   LIN {X 4.730, Y 38.392, Z 10.200} C_DIS
   LIN {X 4.962, Y 37.586, Z 10.200} C_DIS
   LIN {X 5.429, Y 35.866, Z 10.200} C_DIS
   LIN {X 5.472, Y 35.706, Z 10.200} C_DIS
   LIN {X 5.506, Y 35.572, Z 10.200} C_DIS
   LIN {X 6.084, Y 33.263, Z 10.200} C_DIS
   LIN {X 6.346, Y 32.125, Z 10.200} C_DIS
   LIN {X 6.530, Y 31.325, Z 10.200} C_DIS
   LIN {X 7.402, Y 26.882, Z 10.200} C_DIS
   LIN {X 7.443, Y 26.679, Z 10.200} C_DIS
   LIN {X 7.483, Y 26.451, Z 10.200} C_DIS
   LIN {X 7.771, Y 24.714, Z 10.200} C_DIS
   LIN {X 8.198, Y 21.694, Z 10.200} C_DIS
   LIN {X 8.305, Y 20.843, Z 10.200} C_DIS
   LIN {X 8.407, Y 19.968, Z 10.200} C_DIS
   LIN {X 8.478, Y 19.358, Z 10.200} C_DIS
   LIN {X 8.502, Y 19.110, Z 10.200} C_DIS
   LIN {X 8.808, Y 15.682, Z 10.200} C_DIS
   LIN {X 8.841, Y 15.275, Z 10.200} C_DIS
   LIN {X 8.850, Y 15.139, Z 10.200} C_DIS
   LIN {X 8.857, Y 15.004, Z 10.200} C_DIS
   LIN {X 8.864, Y 14.867, Z 10.200} C_DIS
   LIN {X 8.927, Y 13.736, Z 10.200} C_DIS
   LIN {X 9.005, Y 12.397, Z 10.200} C_DIS
   LIN {X 9.017, Y 12.053, Z 10.200} C_DIS
   LIN {X 9.102, Y 8.921, Z 10.200} C_DIS
   LIN {X 9.107, Y 7.373, Z 10.200} C_DIS
   LIN {X 9.109, Y 6.968, Z 10.200} C_DIS
   LIN {X 9.106, Y 6.824, Z 10.200} C_DIS
   LIN {X 9.029, Y 3.343, Z 10.200} C_DIS
   LIN {X 8.935, Y 1.364, Z 10.200} C_DIS
   LIN {X 8.928, Y 1.257, Z 10.200} C_DIS
   LIN {X 8.900, Y 0.914, Z 10.200} C_DIS
   LIN {X 8.633, Y -2.599, Z 10.200} C_DIS
   LIN {X 8.512, Y -3.854, Z 10.200} C_DIS
   LIN {X 8.395, Y -4.942, Z 10.200} C_DIS
   LIN {X 8.356, Y -5.250, Z 10.200} C_DIS
   LIN {X 7.974, Y -8.182, Z 10.200} C_DIS
   LIN {X 7.923, Y -8.524, Z 10.200} C_DIS
   LIN {X 7.807, Y -9.164, Z 10.200} C_DIS
   LIN {X 7.070, Y -13.450, Z 10.200} C_DIS
   LIN {X 6.629, Y -15.636, Z 10.200} C_DIS
   LIN {X 6.073, Y -18.076, Z 10.200} C_DIS
   LIN {X 5.567, Y -20.105, Z 10.200} C_DIS
   LIN {X 5.149, Y -21.676, Z 10.200} C_DIS
   LIN {X 4.625, Y -23.491, Z 10.200} C_DIS
   LIN {X 4.417, Y -24.222, Z 10.200} C_DIS
   LIN {X 4.241, Y -24.798, Z 10.200} C_DIS
   LIN {X 3.838, Y -26.087, Z 10.200} C_DIS
   LIN {X 2.539, Y -28.357, Z 10.200} C_DIS
   LIN {X 1.987, Y -29.326, Z 10.200} C_DIS
   LIN {X 1.547, Y -29.692, Z 10.200} C_DIS
   LIN {X -0.334, Y -31.205, Z 10.200} C_DIS
   LIN {X -2.195, Y -31.910, Z 10.200} C_DIS
   LIN {X -3.063, Y -32.217, Z 10.200} C_DIS
   LIN {X -4.813, Y -32.267, Z 10.200} C_DIS
   LIN {X -5.950, Y -32.313, Z 10.200} C_DIS
   LIN {X -6.218, Y -32.259, Z 10.200} C_DIS
   LIN {X -6.409, Y -32.191, Z 10.200} C_DIS
   LIN {X -9.906, Y -30.751, Z 10.200} C_DIS
   LIN {X -10.167, Y -30.607, Z 10.200} C_DIS
   LIN {X -10.841, Y -30.035, Z 10.200} C_DIS
   LIN {X -11.131, Y -29.776, Z 10.200} C_DIS
   LIN {X -11.194, Y -29.687, Z 10.200} C_DIS
   LIN {X -11.449, Y -29.321, Z 10.200} C_DIS
   LIN {X -12.804, Y -27.467, Z 10.200} C_DIS
   LIN {X -13.363, Y -25.694, Z 10.200} C_DIS
   LIN {X -13.691, Y -24.527, Z 10.200} C_DIS
   LIN {X -13.623, Y -23.242, Z 10.200} C_DIS
   LIN {X -13.562, Y -21.557, Z 10.200} C_DIS
   LIN {X -12.981, Y -20.117, Z 10.200} C_DIS
   LIN {X -12.370, Y -18.619, Z 10.200} C_DIS
   LIN {X -11.694, Y -17.504, Z 10.200} C_DIS
   LIN {X -10.729, Y -15.883, Z 10.200} C_DIS
   LIN {X -8.996, Y -12.598, Z 10.200} C_DIS
   LIN {X -8.678, Y -12.002, Z 10.200} C_DIS
   LIN {X -8.590, Y -11.835, Z 10.200} C_DIS
   LIN {X -8.537, Y -11.731, Z 10.200} C_DIS
   LIN {X -7.939, Y -10.386, Z 10.200} C_DIS
   LIN {X -6.633, Y -7.473, Z 10.200} C_DIS
   LIN {X -6.291, Y -6.580, Z 10.200} C_DIS
   LIN {X -5.258, Y -3.854, Z 10.200} C_DIS
   LIN {X -4.877, Y -2.572, Z 10.200}
   LaserEnd_Ext()
   LIN {X -0.927, Y -30.360, Z 10.200}
   LaserStart_Ext()
   LIN {X -8.228, Y -30.360, Z 10.200}
   LaserEnd_Ext()
   LIN {X -10.092, Y -29.360, Z 10.200}
   LaserStart_Ext()
   LIN {X 0.364, Y -29.360, Z 10.200}
   LaserEnd_Ext()
   LIN {X 1.386, Y -28.360, Z 10.200}
   LaserStart_Ext()
   LIN {X -10.912, Y -28.360, Z 10.200}
   LaserEnd_Ext()
   LIN {X -11.643, Y -27.360, Z 10.200}
   LaserStart_Ext()
   LIN {X 1.957, Y -27.360, Z 10.200}
   LaserEnd_Ext()
   LIN {X 2.530, Y -26.360, Z 10.200}
   LaserStart_Ext()
   LIN {X -12.104, Y -26.360, Z 10.200}
   LaserEnd_Ext()
   LIN {X -12.418, Y -25.360, Z 10.200}
   LaserStart_Ext()
   LIN {X -5.393, Y -25.360, Z 10.200}
   LaserEnd_Ext()
   LIN {X -4.055, Y -25.360, Z 10.200}
   LaserStart_Ext()
   LIN {X 3.018, Y -25.360, Z 10.200}
   LaserEnd_Ext()
   LIN {X 3.329, Y -24.360, Z 10.200}
   LaserStart_Ext()
   LIN {X -2.856, Y -24.360, Z 10.200}
   LaserEnd_Ext()
   LIN {X -6.619, Y -24.360, Z 10.200}
   LaserStart_Ext()
   LIN {X -12.681, Y -24.360, Z 10.200}
   LaserEnd_Ext()
   LIN {X -12.628, Y -23.360, Z 10.200}
   LaserStart_Ext()
   LIN {X -6.894, Y -23.360, Z 10.200}
   LaserEnd_Ext()
   LIN {X -2.671, Y -23.360, Z 10.200}
   LaserStart_Ext()
   LIN {X 3.623, Y -23.360, Z 10.200}
   LaserEnd_Ext()
   LIN {X 3.911, Y -22.360, Z 10.200}
   LaserStart_Ext()
   LIN {X -2.769, Y -22.360, Z 10.200}
   LaserEnd_Ext()
   LIN {X -6.651, Y -22.360, Z 10.200}
   LaserStart_Ext()
   LIN {X -12.591, Y -22.360, Z 10.200}
   LaserEnd_Ext()
   LIN {X -12.405, Y -21.360, Z 10.200}
   LaserStart_Ext()
   LIN {X -5.680, Y -21.360, Z 10.200}
   LaserEnd_Ext()
   LIN {X -3.731, Y -21.360, Z 10.200}
   LaserStart_Ext()
   LIN {X 4.199, Y -21.360, Z 10.200}
   LaserEnd_Ext()
   LIN {X 4.464, Y -20.360, Z 10.200}
   LaserStart_Ext()
   LIN {X -12.000, Y -20.360, Z 10.200}
   LaserEnd_Ext()
   LIN {X -11.592, Y -19.360, Z 10.200}
   LaserStart_Ext()
   LIN {X 4.722, Y -19.360, Z 10.200}
   LaserEnd_Ext()
   LIN {X 4.972, Y -18.360, Z 10.200}
   LaserStart_Ext()
   LIN {X -11.044, Y -18.360, Z 10.200}
   LaserEnd_Ext()
   LIN {X -10.445, Y -17.360, Z 10.200}
   LaserStart_Ext()
   LIN {X 5.211, Y -17.360, Z 10.200}
   LaserEnd_Ext()
   LIN {X 5.439, Y -16.360, Z 10.200}
   LaserStart_Ext()
   LIN {X -9.851, Y -16.360, Z 10.200}
   LaserEnd_Ext()
   LIN {X -9.323, Y -15.360, Z 10.200}
   LaserStart_Ext()
   LIN {X 5.665, Y -15.360, Z 10.200}
   LaserEnd_Ext()
   LIN {X 5.866, Y -14.360, Z 10.200}
   LaserStart_Ext()
   LIN {X -8.795, Y -14.360, Z 10.200}
   LaserEnd_Ext()
   LIN {X -8.268, Y -13.360, Z 10.200}
   LaserStart_Ext()
   LIN {X 6.068, Y -13.360, Z 10.200}
   LaserEnd_Ext()
   LIN {X 6.243, Y -12.360, Z 10.200}
   LaserStart_Ext()
   LIN {X -7.736, Y -12.360, Z 10.200}
   LaserEnd_Ext()
   LIN {X -7.277, Y -11.360, Z 10.200}
   LaserStart_Ext()
   LIN {X 6.415, Y -11.360, Z 10.200}
   LaserEnd_Ext()
   LIN {X 6.587, Y -10.360, Z 10.200}
   LaserStart_Ext()
   LIN {X -6.831, Y -10.360, Z 10.200}
   LaserEnd_Ext()
   LIN {X -6.383, Y -9.360, Z 10.200}
   LaserStart_Ext()
   LIN {X 6.758, Y -9.360, Z 10.200}
   LaserEnd_Ext()
   LIN {X 6.937, Y -8.360, Z 10.200}
   LaserStart_Ext()
   LIN {X -5.935, Y -8.360, Z 10.200}
   LaserEnd_Ext()
   LIN {X -5.519, Y -7.360, Z 10.200}
   LaserStart_Ext()
   LIN {X 7.073, Y -7.360, Z 10.200}
   LaserEnd_Ext()
   LIN {X 7.203, Y -6.360, Z 10.200}
   LaserStart_Ext()
   LIN {X -5.138, Y -6.360, Z 10.200}
   LaserEnd_Ext()
   LIN {X -4.760, Y -5.360, Z 10.200}
   LaserStart_Ext()
   LIN {X 7.333, Y -5.360, Z 10.200}
   LaserEnd_Ext()
   LIN {X 7.452, Y -4.360, Z 10.200}
   LaserStart_Ext()
   LIN {X -4.381, Y -4.360, Z 10.200}
   LaserEnd_Ext()
   LIN {X -4.068, Y -3.360, Z 10.200}
   LaserStart_Ext()
   LIN {X 7.555, Y -3.360, Z 10.200}
   LaserEnd_Ext()
   LIN {X 7.648, Y -2.360, Z 10.200}
   LaserStart_Ext()
   LIN {X -3.759, Y -2.360, Z 10.200}
   LaserEnd_Ext()
   LIN {X -3.437, Y -1.360, Z 10.200}
   LaserStart_Ext()
   LIN {X 7.724, Y -1.360, Z 10.200}
   LaserEnd_Ext()
   LIN {X 7.800, Y -0.360, Z 10.200}
   LaserStart_Ext()
   LIN {X -3.115, Y -0.360, Z 10.200}
   LaserEnd_Ext()
   LIN {X -2.824, Y 0.640, Z 10.200}
   LaserStart_Ext()
   LIN {X 7.876, Y 0.640, Z 10.200}
   LaserEnd_Ext()
   LIN {X 7.947, Y 1.640, Z 10.200}
   LaserStart_Ext()
   LIN {X -2.546, Y 1.640, Z 10.200}
   LaserEnd_Ext()
   LIN {X -2.297, Y 2.640, Z 10.200}
   LaserStart_Ext()
   LIN {X 7.994, Y 2.640, Z 10.200}
   LaserEnd_Ext()
   LIN {X 8.035, Y 3.640, Z 10.200}
   LaserStart_Ext()
   LIN {X -2.063, Y 3.640, Z 10.200}
   LaserEnd_Ext()
   LIN {X -1.857, Y 4.640, Z 10.200}
   LaserStart_Ext()
   LIN {X 8.057, Y 4.640, Z 10.200}
   LaserEnd_Ext()
   LIN {X 8.080, Y 5.640, Z 10.200}
   LaserStart_Ext()
   LIN {X -1.653, Y 5.640, Z 10.200}
   LaserEnd_Ext()
   LIN {X -1.438, Y 6.640, Z 10.200}
   LaserStart_Ext()
   LIN {X 8.102, Y 6.640, Z 10.200}
   LaserEnd_Ext()
   LIN {X 8.107, Y 7.640, Z 10.200}
   LaserStart_Ext()
   LIN {X -1.262, Y 7.640, Z 10.200}
   LaserEnd_Ext()
   LIN {X -1.098, Y 8.640, Z 10.200}
   LaserStart_Ext()
   LIN {X 8.103, Y 8.640, Z 10.200}
   LaserEnd_Ext()
   LIN {X 8.083, Y 9.640, Z 10.200}
   LaserStart_Ext()
   LIN {X -0.945, Y 9.640, Z 10.200}
   LaserEnd_Ext()
   LIN {X -0.820, Y 10.640, Z 10.200}
   LaserStart_Ext()
   LIN {X 8.055, Y 10.640, Z 10.200}
   LaserEnd_Ext()
   LIN {X 8.028, Y 11.640, Z 10.200}
   LaserStart_Ext()
   LIN {X -0.695, Y 11.640, Z 10.200}
   LaserEnd_Ext()
   LIN {X -0.574, Y 12.640, Z 10.200}
   LaserStart_Ext()
   LIN {X 7.989, Y 12.640, Z 10.200}
   LaserEnd_Ext()
   LIN {X 7.931, Y 13.640, Z 10.200}
   LaserStart_Ext()
   LIN {X -0.496, Y 13.640, Z 10.200}
   LaserEnd_Ext()
   LIN {X -0.418, Y 14.640, Z 10.200}
   LaserStart_Ext()
   LIN {X 7.875, Y 14.640, Z 10.200}
   LaserEnd_Ext()
   LIN {X 7.808, Y 15.640, Z 10.200}
   LaserStart_Ext()
   LIN {X -0.340, Y 15.640, Z 10.200}
   LaserEnd_Ext()
   LIN {X -0.276, Y 16.640, Z 10.200}
   LaserStart_Ext()
   LIN {X 7.719, Y 16.640, Z 10.200}
   LaserEnd_Ext()
   LIN {X 7.630, Y 17.640, Z 10.200}
   LaserStart_Ext()
   LIN {X -0.236, Y 17.640, Z 10.200}
   LaserEnd_Ext()
   LIN {X -0.209, Y 18.640, Z 10.200}
   LaserStart_Ext()
   LIN {X 7.540, Y 18.640, Z 10.200}
   LaserEnd_Ext()
   LIN {X 7.439, Y 19.640, Z 10.200}
   LaserStart_Ext()
   LIN {X -0.198, Y 19.640, Z 10.200}
   LaserEnd_Ext()
   LIN {X -0.205, Y 20.640, Z 10.200}
   LaserStart_Ext()
   LIN {X 7.322, Y 20.640, Z 10.200}
   LaserEnd_Ext()
   LIN {X 7.195, Y 21.640, Z 10.200}
   LaserStart_Ext()
   LIN {X -0.229, Y 21.640, Z 10.200}
   LaserEnd_Ext()
   LIN {X -0.254, Y 22.640, Z 10.200}
   LaserStart_Ext()
   LIN {X 7.054, Y 22.640, Z 10.200}
   LaserEnd_Ext()
   LIN {X 6.913, Y 23.640, Z 10.200}
   LaserStart_Ext()
   LIN {X -0.278, Y 23.640, Z 10.200}
   LaserEnd_Ext()
   LIN {X -0.333, Y 24.640, Z 10.200}
   LaserStart_Ext()
   LIN {X 6.769, Y 24.640, Z 10.200}
   LaserEnd_Ext()
   LIN {X 6.604, Y 25.640, Z 10.200}
   LaserStart_Ext()
   LIN {X -0.404, Y 25.640, Z 10.200}
   LaserEnd_Ext()
   LIN {X -0.489, Y 26.640, Z 10.200}
   LaserStart_Ext()
   LIN {X 6.431, Y 26.640, Z 10.200}
   LaserEnd_Ext()
   LIN {X 6.234, Y 27.640, Z 10.200}
   LaserStart_Ext()
   LIN {X -0.590, Y 27.640, Z 10.200}
   LaserEnd_Ext()
   LIN {X -0.692, Y 28.640, Z 10.200}
   LaserStart_Ext()
   LIN {X 6.038, Y 28.640, Z 10.200}
   LaserEnd_Ext()
   LIN {X 5.842, Y 29.640, Z 10.200}
   LaserStart_Ext()
   LIN {X -0.813, Y 29.640, Z 10.200}
   LaserEnd_Ext()
   LIN {X -0.956, Y 30.640, Z 10.200}
   LaserStart_Ext()
   LIN {X 5.646, Y 30.640, Z 10.200}
   LaserEnd_Ext()
   LIN {X 5.431, Y 31.640, Z 10.200}
   LaserStart_Ext()
   LIN {X -1.099, Y 31.640, Z 10.200}
   LaserEnd_Ext()
   LIN {X -1.261, Y 32.640, Z 10.200}
   LaserStart_Ext()
   LIN {X 5.201, Y 32.640, Z 10.200}
   LaserEnd_Ext()
   LIN {X 4.959, Y 33.640, Z 10.200}
   LaserStart_Ext()
   LIN {X -1.441, Y 33.640, Z 10.200}
   LaserEnd_Ext()
   LIN {X -1.627, Y 34.640, Z 10.200}
   LaserStart_Ext()
   LIN {X 4.709, Y 34.640, Z 10.200}
   LaserEnd_Ext()
   LIN {X 4.454, Y 35.640, Z 10.200}
   LaserStart_Ext()
   LIN {X -1.836, Y 35.640, Z 10.200}
   LaserEnd_Ext()
   LIN {X -2.052, Y 36.640, Z 10.200}
   LaserStart_Ext()
   LIN {X 4.182, Y 36.640, Z 10.200}
   LaserEnd_Ext()
   LIN {X 3.906, Y 37.640, Z 10.200}
   LaserStart_Ext()
   LIN {X -2.199, Y 37.640, Z 10.200}
   LaserEnd_Ext()
   LIN {X -2.148, Y 38.640, Z 10.200}
   LaserStart_Ext()
   LIN {X 3.617, Y 38.640, Z 10.200}
   LaserEnd_Ext()
   LIN {X 3.121, Y 39.640, Z 10.200}
   LaserStart_Ext()
   LIN {X -1.702, Y 39.640, Z 10.200}
   LaserEnd_Ext()
   LIN {X -0.132, Y 40.640, Z 10.200}
   LaserStart_Ext()
   LIN {X 1.883, Y 40.640, Z 10.200}
   LaserEnd_Ext()
   LIN {X -6.268, Y -21.991, Z 11.050}
   LaserStart_Ext()
   LIN {X -6.676, Y -23.129, Z 11.050} C_DIS
   LIN {X -6.630, Y -23.393, Z 11.050} C_DIS
   LIN {X -6.422, Y -24.182, Z 11.050} C_DIS
   LIN {X -6.288, Y -24.390, Z 11.050} C_DIS
   LIN {X -6.019, Y -24.701, Z 11.050} C_DIS
   LIN {X -5.700, Y -24.925, Z 11.050} C_DIS
   LIN {X -5.541, Y -25.028, Z 11.050} C_DIS
   LIN {X -5.254, Y -25.113, Z 11.050} C_DIS
   LIN {X -4.893, Y -25.217, Z 11.050} C_DIS
   LIN {X -4.115, Y -25.153, Z 11.050} C_DIS
   LIN {X -3.320, Y -24.726, Z 11.050} C_DIS
   LIN {X -2.743, Y -23.895, Z 11.050} C_DIS
   LIN {X -2.646, Y -22.978, Z 11.050} C_DIS
   LIN {X -2.635, Y -22.876, Z 11.050} C_DIS
   LIN {X -2.683, Y -22.714, Z 11.050} C_DIS
   LIN {X -2.799, Y -22.327, Z 11.050} C_DIS
   LIN {X -2.978, Y -22.045, Z 11.050} C_DIS
   LIN {X -3.106, Y -21.854, Z 11.050} C_DIS
   LIN {X -3.553, Y -21.505, Z 11.050} C_DIS
   LIN {X -3.707, Y -21.381, Z 11.050} C_DIS
   LIN {X -3.910, Y -21.327, Z 11.050} C_DIS
   LIN {X -4.518, Y -21.162, Z 11.050} C_DIS
   LIN {X -4.733, Y -21.182, Z 11.050} C_DIS
   LIN {X -5.193, Y -21.239, Z 11.050} C_DIS
   LIN {X -6.249, Y -21.966, Z 11.050} C_DIS
   LIN {X -6.268, Y -21.991, Z 11.050}
   LaserEnd_Ext()
   LIN {X -1.587, Y 27.145, Z 11.050}
   LaserStart_Ext()
   LIN {X -1.698, Y 28.227, Z 11.050} C_DIS
   LIN {X -1.788, Y 29.112, Z 11.050} C_DIS
   LIN {X -1.997, Y 30.562, Z 11.050} C_DIS
   LIN {X -2.204, Y 31.978, Z 11.050} C_DIS
   LIN {X -2.451, Y 33.326, Z 11.050} C_DIS
   LIN {X -2.629, Y 34.311, Z 11.050} C_DIS
   LIN {X -2.716, Y 34.727, Z 11.050} C_DIS
   LIN {X -2.959, Y 35.877, Z 11.050} C_DIS
   LIN {X -3.169, Y 36.818, Z 11.050} C_DIS
   LIN {X -3.233, Y 37.099, Z 11.050} C_DIS
   LIN {X -3.257, Y 37.673, Z 11.050} C_DIS
   LIN {X -3.305, Y 38.649, Z 11.050} C_DIS
   LIN {X -3.053, Y 39.374, Z 11.050} C_DIS
   LIN {X -2.780, Y 40.095, Z 11.050} C_DIS
   LIN {X -2.141, Y 40.740, Z 11.050} C_DIS
   LIN {X -1.529, Y 41.382, Z 11.050} C_DIS
   LIN {X -0.612, Y 41.638, Z 11.050} C_DIS
   LIN {X 0.767, Y 42.010, Z 11.050} C_DIS
   LIN {X 1.941, Y 41.701, Z 11.050} C_DIS
   LIN {X 2.458, Y 41.562, Z 11.050} C_DIS
   LIN {X 3.056, Y 41.061, Z 11.050} C_DIS
   LIN {X 3.795, Y 40.443, Z 11.050} C_DIS
   LIN {X 4.094, Y 39.860, Z 11.050} C_DIS
   LIN {X 4.465, Y 39.130, Z 11.050} C_DIS
   LIN {X 4.760, Y 38.111, Z 11.050} C_DIS
   LIN {X 4.902, Y 37.627, Z 11.050} C_DIS
   LIN {X 5.021, Y 37.196, Z 11.050} C_DIS
   LIN {X 5.420, Y 35.738, Z 11.050} C_DIS
   LIN {X 5.963, Y 33.578, Z 11.050} C_DIS
   LIN {X 6.076, Y 33.126, Z 11.050} C_DIS
   LIN {X 6.235, Y 32.437, Z 11.050} C_DIS
   LIN {X 6.550, Y 31.068, Z 11.050} C_DIS
   LIN {X 7.293, Y 27.283, Z 11.050} C_DIS
   LIN {X 7.468, Y 26.385, Z 11.050} C_DIS
   LIN {X 7.598, Y 25.570, Z 11.050} C_DIS
   LIN {X 7.815, Y 24.263, Z 11.050} C_DIS
   LIN {X 8.099, Y 22.252, Z 11.050} C_DIS
   LIN {X 8.363, Y 20.166, Z 11.050} C_DIS
   LIN {X 8.494, Y 19.041, Z 11.050} C_DIS
   LIN {X 8.820, Y 15.370, Z 11.050} C_DIS
   LIN {X 8.855, Y 14.892, Z 11.050} C_DIS
   LIN {X 8.997, Y 12.432, Z 11.050} C_DIS
   LIN {X 9.035, Y 11.400, Z 11.050} C_DIS
   LIN {X 9.101, Y 8.956, Z 11.050} C_DIS
   LIN {X 9.107, Y 7.334, Z 11.050} C_DIS
   LIN {X 9.109, Y 6.597, Z 11.050} C_DIS
   LIN {X 9.043, Y 3.619, Z 11.050} C_DIS
   LIN {X 9.029, Y 3.109, Z 11.050} C_DIS
   LIN {X 8.952, Y 1.501, Z 11.050} C_DIS
   LIN {X 8.905, Y 0.693, Z 11.050} C_DIS
   LIN {X 8.689, Y -2.135, Z 11.050} C_DIS
   LIN {X 8.448, Y -4.657, Z 11.050} C_DIS
   LIN {X 8.424, Y -4.872, Z 11.050} C_DIS
   LIN {X 8.310, Y -5.755, Z 11.050} C_DIS
   LIN {X 7.991, Y -8.255, Z 11.050} C_DIS
   LIN {X 7.835, Y -9.263, Z 11.050} C_DIS
   LIN {X 7.198, Y -12.969, Z 11.050} C_DIS
   LIN {X 6.519, Y -16.333, Z 11.050} C_DIS
   LIN {X 6.216, Y -17.665, Z 11.050} C_DIS
   LIN {X 5.381, Y -21.013, Z 11.050} C_DIS
   LIN {X 5.245, Y -21.523, Z 11.050} C_DIS
   LIN {X 5.075, Y -22.112, Z 11.050} C_DIS
   LIN {X 4.493, Y -24.156, Z 11.050} C_DIS
   LIN {X 4.002, Y -25.765, Z 11.050} C_DIS
   LIN {X 3.921, Y -26.025, Z 11.050} C_DIS
   LIN {X 3.659, Y -26.483, Z 11.050} C_DIS
   LIN {X 2.075, Y -29.266, Z 11.050} C_DIS
   LIN {X 0.809, Y -30.317, Z 11.050} C_DIS
   LIN {X -0.198, Y -31.127, Z 11.050} C_DIS
   LIN {X -2.516, Y -32.005, Z 11.050} C_DIS
   LIN {X -2.875, Y -32.148, Z 11.050} C_DIS
   LIN {X -3.148, Y -32.175, Z 11.050} C_DIS
   LIN {X -5.770, Y -32.280, Z 11.050} C_DIS
   LIN {X -6.545, Y -32.125, Z 11.050} C_DIS
   LIN {X -7.097, Y -31.928, Z 11.050} C_DIS
   LIN {X -9.327, Y -31.010, Z 11.050} C_DIS
   LIN {X -9.944, Y -30.671, Z 11.050} C_DIS
   LIN {X -10.472, Y -30.223, Z 11.050} C_DIS
   LIN {X -10.975, Y -29.813, Z 11.050} C_DIS
   LIN {X -11.154, Y -29.620, Z 11.050} C_DIS
   LIN {X -11.482, Y -29.153, Z 11.050} C_DIS
   LIN {X -12.688, Y -27.503, Z 11.050} C_DIS
   LIN {X -13.496, Y -24.937, Z 11.050} C_DIS
   LIN {X -13.597, Y -24.641, Z 11.050} C_DIS
   LIN {X -13.595, Y -24.371, Z 11.050} C_DIS
   LIN {X -13.492, Y -21.533, Z 11.050} C_DIS
   LIN {X -12.309, Y -18.605, Z 11.050} C_DIS
   LIN {X -10.673, Y -15.853, Z 11.050} C_DIS
   LIN {X -9.083, Y -12.840, Z 11.050} C_DIS
   LIN {X -8.631, Y -11.983, Z 11.050} C_DIS
   LIN {X -8.372, Y -11.427, Z 11.050} C_DIS
   LIN {X -6.783, Y -7.883, Z 11.050} C_DIS
   LIN {X -6.017, Y -5.881, Z 11.050} C_DIS
   LIN {X -5.215, Y -3.764, Z 11.050} C_DIS
   LIN {X -4.457, Y -1.215, Z 11.050} C_DIS
   LIN {X -3.867, Y 0.618, Z 11.050} C_DIS
   LIN {X -3.554, Y 1.723, Z 11.050} C_DIS
   LIN {X -3.290, Y 2.781, Z 11.050} C_DIS
   LIN {X -3.188, Y 3.239, Z 11.050} C_DIS
   LIN {X -2.871, Y 4.788, Z 11.050} C_DIS
   LIN {X -2.413, Y 6.861, Z 11.050} C_DIS
   LIN {X -2.071, Y 8.916, Z 11.050} C_DIS
   LIN {X -1.996, Y 9.426, Z 11.050} C_DIS
   LIN {X -1.613, Y 12.426, Z 11.050} C_DIS
   LIN {X -1.540, Y 13.310, Z 11.050} C_DIS
   LIN {X -1.323, Y 16.095, Z 11.050} C_DIS
   LIN {X -1.299, Y 16.648, Z 11.050} C_DIS
   LIN {X -1.268, Y 17.324, Z 11.050} C_DIS
   LIN {X -1.243, Y 18.170, Z 11.050} C_DIS
   LIN {X -1.231, Y 19.188, Z 11.050} C_DIS
   LIN {X -1.229, Y 20.623, Z 11.050} C_DIS
   LIN {X -1.294, Y 23.277, Z 11.050} C_DIS
   LIN {X -1.341, Y 24.101, Z 11.050} C_DIS
   LIN {X -1.403, Y 24.943, Z 11.050} C_DIS
   LIN {X -1.463, Y 25.994, Z 11.050} C_DIS
   LIN {X -1.552, Y 26.799, Z 11.050} C_DIS
   LIN {X -1.587, Y 27.145, Z 11.050}
   LaserEnd_Ext()
   LIN {X 7.602, Y -3.000, Z 11.050}
   LaserStart_Ext()
   LIN {X 7.602, Y 17.784, Z 11.050}
   LaserEnd_Ext()
   LIN {X 6.602, Y 25.467, Z 11.050}
   LaserStart_Ext()
   LIN {X 6.602, Y -10.533, Z 11.050}
   LaserEnd_Ext()
   LIN {X 5.602, Y -15.824, Z 11.050}
   LaserStart_Ext()
   LIN {X 5.602, Y 30.708, Z 11.050}
   LaserEnd_Ext()
   LIN {X 4.602, Y 34.889, Z 11.050}
   LaserStart_Ext()
   LIN {X 4.602, Y -20.003, Z 11.050}
   LaserEnd_Ext()
   LIN {X 3.602, Y -23.634, Z 11.050}
   LaserStart_Ext()
   LIN {X 3.602, Y 38.515, Z 11.050}
   LaserEnd_Ext()
   LIN {X 2.602, Y 40.137, Z 11.050}
   LaserStart_Ext()
   LIN {X 2.602, Y -26.318, Z 11.050}
   LaserEnd_Ext()
   LIN {X 1.602, Y -28.076, Z 11.050}
   LaserStart_Ext()
   LIN {X 1.602, Y 40.756, Z 11.050}
   LaserEnd_Ext()
   LIN {X 0.602, Y 40.930, Z 11.050}
   LaserStart_Ext()
   LIN {X 0.602, Y -29.189, Z 11.050}
   LaserEnd_Ext()
   LIN {X -0.398, Y -30.005, Z 11.050}
   LaserStart_Ext()
   LIN {X -0.398, Y 15.098, Z 11.050}
   LaserEnd_Ext()
   LIN {X -0.398, Y 24.916, Z 11.050}
   LaserStart_Ext()
   LIN {X -0.398, Y 40.660, Z 11.050}
   LaserEnd_Ext()
   LIN {X -1.398, Y 40.070, Z 11.050}
   LaserStart_Ext()
   LIN {X -1.398, Y 33.127, Z 11.050}
   LaserEnd_Ext()
   LIN {X -1.398, Y 6.871, Z 11.050}
   LaserStart_Ext()
   LIN {X -1.398, Y -30.512, Z 11.050}
   LaserEnd_Ext()
   LIN {X -2.398, Y -30.891, Z 11.050}
   LaserStart_Ext()
   LIN {X -2.398, Y -25.160, Z 11.050}
   LaserEnd_Ext()
   LIN {X -2.398, Y -21.150, Z 11.050}
   LaserStart_Ext()
   LIN {X -2.398, Y 2.224, Z 11.050}
   LaserEnd_Ext()
   LIN {X -3.398, Y -1.188, Z 11.050}
   LaserStart_Ext()
   LIN {X -3.398, Y -20.432, Z 11.050}
   LaserEnd_Ext()
   LIN {X -3.398, Y -25.908, Z 11.050}
   LaserStart_Ext()
   LIN {X -3.398, Y -31.184, Z 11.050}
   LaserEnd_Ext()
   LIN {X -4.398, Y -31.224, Z 11.050}
   LaserStart_Ext()
   LIN {X -4.398, Y -26.180, Z 11.050}
   LaserEnd_Ext()
   LIN {X -4.398, Y -20.171, Z 11.050}
   LaserStart_Ext()
   LIN {X -4.398, Y -4.430, Z 11.050}
   LaserEnd_Ext()
   LIN {X -5.398, Y -7.062, Z 11.050}
   LaserStart_Ext()
   LIN {X -5.398, Y -20.261, Z 11.050}
   LaserEnd_Ext()
   LIN {X -5.398, Y -26.112, Z 11.050}
   LaserStart_Ext()
   LIN {X -5.398, Y -31.265, Z 11.050}
   LaserEnd_Ext()
   LIN {X -6.398, Y -31.116, Z 11.050}
   LaserStart_Ext()
   LIN {X -6.398, Y -25.657, Z 11.050}
   LaserEnd_Ext()
   LIN {X -6.398, Y -20.855, Z 11.050}
   LaserStart_Ext()
   LIN {X -6.398, Y -9.469, Z 11.050}
   LaserEnd_Ext()
   LIN {X -7.398, Y -11.700, Z 11.050}
   LaserStart_Ext()
   LIN {X -7.398, Y -22.180, Z 11.050}
   LaserEnd_Ext()
   LIN {X -7.398, Y -24.402, Z 11.050}
   LaserStart_Ext()
   LIN {X -7.398, Y -30.723, Z 11.050}
   LaserEnd_Ext()
   LIN {X -8.398, Y -30.311, Z 11.050}
   LaserStart_Ext()
   LIN {X -8.398, Y -13.685, Z 11.050}
   LaserEnd_Ext()
   LIN {X -9.398, Y -15.580, Z 11.050}
   LaserStart_Ext()
   LIN {X -9.398, Y -29.823, Z 11.050}
   LaserEnd_Ext()
   LIN {X -10.398, Y -28.957, Z 11.050}
   LaserStart_Ext()
   LIN {X -10.398, Y -17.346, Z 11.050}
   LaserEnd_Ext()
   LIN {X -11.398, Y -19.026, Z 11.050}
   LaserStart_Ext()
   LIN {X -11.398, Y -27.573, Z 11.050}
   LaserEnd_Ext()
   LIN {X -12.398, Y -25.095, Z 11.050}
   LaserStart_Ext()
   LIN {X -12.398, Y -21.495, Z 11.050}
   LaserEnd_Ext()
   LIN {X -4.864, Y -25.940, Z 11.900}
   LaserStart_Ext()
   LIN {X -4.243, Y -25.966, Z 11.900} C_DIS
   LIN {X -4.008, Y -25.904, Z 11.900} C_DIS
   LIN {X -3.329, Y -25.702, Z 11.900} C_DIS
   LIN {X -3.119, Y -25.586, Z 11.900} C_DIS
   LIN {X -2.544, Y -24.979, Z 11.900} C_DIS
   LIN {X -1.792, Y -23.871, Z 11.900} C_DIS
   LIN {X -1.766, Y -22.530, Z 11.900} C_DIS
   LIN {X -1.786, Y -22.242, Z 11.900} C_DIS
   LIN {X -1.841, Y -22.124, Z 11.900} C_DIS
   LIN {X -2.889, Y -20.825, Z 11.900} C_DIS
   LIN {X -3.228, Y -20.512, Z 11.900} C_DIS
   LIN {X -3.658, Y -20.387, Z 11.900} C_DIS
   LIN {X -4.266, Y -20.212, Z 11.900} C_DIS
   LIN {X -4.841, Y -20.232, Z 11.900} C_DIS
   LIN {X -5.041, Y -20.247, Z 11.900} C_DIS
   LIN {X -6.009, Y -20.665, Z 11.900} C_DIS
   LIN {X -6.432, Y -20.929, Z 11.900} C_DIS
   LIN {X -7.154, Y -21.901, Z 11.900} C_DIS
   LIN {X -7.307, Y -22.360, Z 11.900} C_DIS
   LIN {X -7.427, Y -23.298, Z 11.900} C_DIS
   LIN {X -6.885, Y -24.784, Z 11.900} C_DIS
   LIN {X -6.758, Y -24.954, Z 11.900} C_DIS
   LIN {X -6.304, Y -25.406, Z 11.900} C_DIS
   LIN {X -6.136, Y -25.512, Z 11.900} C_DIS
   LIN {X -5.822, Y -25.701, Z 11.900} C_DIS
   LIN {X -5.240, Y -25.896, Z 11.900} C_DIS
   LIN {X -5.125, Y -25.932, Z 11.900} C_DIS
   LIN {X -4.864, Y -25.940, Z 11.900}
   LaserEnd_Ext()
   LIN {X 5.376, Y 35.731, Z 11.900}
   LaserStart_Ext()
   LIN {X 4.835, Y 37.695, Z 11.900} C_DIS
   LIN {X 4.532, Y 38.730, Z 11.900} C_DIS
   LIN {X 4.395, Y 39.196, Z 11.900} C_DIS
   LIN {X 4.136, Y 39.699, Z 11.900} C_DIS
   LIN {X 3.722, Y 40.508, Z 11.900} C_DIS
   LIN {X 3.043, Y 41.075, Z 11.900} C_DIS
   LIN {X 2.382, Y 41.624, Z 11.900} C_DIS
   LIN {X 0.705, Y 42.063, Z 11.900} C_DIS
   LIN {X -1.632, Y 41.413, Z 11.900} C_DIS
   LIN {X -2.238, Y 40.795, Z 11.900} C_DIS
   LIN {X -2.800, Y 40.229, Z 11.900} C_DIS
   LIN {X -3.058, Y 39.545, Z 11.900} C_DIS
   LIN {X -3.374, Y 38.685, Z 11.900} C_DIS
   LIN {X -3.345, Y 38.254, Z 11.900} C_DIS
   LIN {X -3.298, Y 37.147, Z 11.900} C_DIS
   LIN {X -3.049, Y 36.049, Z 11.900} C_DIS
   LIN {X -3.022, Y 35.926, Z 11.900} C_DIS
   LIN {X -2.957, Y 35.617, Z 11.900} C_DIS
   LIN {X -2.688, Y 34.360, Z 11.900} C_DIS
   LIN {X -2.390, Y 32.749, Z 11.900} C_DIS
   LIN {X -2.258, Y 32.028, Z 11.900} C_DIS
   LIN {X -2.101, Y 30.957, Z 11.900} C_DIS
   LIN {X -1.835, Y 29.163, Z 11.900} C_DIS
   LIN {X -1.715, Y 27.989, Z 11.900} C_DIS
   LIN {X -1.652, Y 27.374, Z 11.900} C_DIS
   LIN {X -1.493, Y 25.938, Z 11.900} C_DIS
   LIN {X -1.386, Y 24.063, Z 11.900} C_DIS
   LIN {X -1.343, Y 23.467, Z 11.900} C_DIS
   LIN {X -1.309, Y 22.883, Z 11.900} C_DIS
   LIN {X -1.263, Y 21.005, Z 11.900} C_DIS
   LIN {X -1.267, Y 18.546, Z 11.900} C_DIS
   LIN {X -1.275, Y 17.869, Z 11.900} C_DIS
   LIN {X -1.292, Y 17.306, Z 11.900} C_DIS
   LIN {X -1.312, Y 16.856, Z 11.900} C_DIS
   LIN {X -1.353, Y 15.914, Z 11.900} C_DIS
   LIN {X -1.512, Y 13.879, Z 11.900} C_DIS
   LIN {X -1.647, Y 12.244, Z 11.900} C_DIS
   LIN {X -1.932, Y 10.004, Z 11.900} C_DIS
   LIN {X -2.207, Y 8.153, Z 11.900} C_DIS
   LIN {X -2.446, Y 6.715, Z 11.900} C_DIS
   LIN {X -3.187, Y 3.358, Z 11.900} C_DIS
   LIN {X -3.357, Y 2.528, Z 11.900} C_DIS
   LIN {X -3.412, Y 2.283, Z 11.900} C_DIS
   LIN {X -3.553, Y 1.716, Z 11.900} C_DIS
   LIN {X -3.721, Y 1.124, Z 11.900} C_DIS
   LIN {X -4.037, Y 0.141, Z 11.900} C_DIS
   LIN {X -5.172, Y -3.675, Z 11.900} C_DIS
   LIN {X -5.743, Y -5.182, Z 11.900} C_DIS
   LIN {X -6.933, Y -8.292, Z 11.900} C_DIS
   LIN {X -8.083, Y -10.857, Z 11.900} C_DIS
   LIN {X -8.742, Y -12.268, Z 11.900} C_DIS
   LIN {X -9.889, Y -14.445, Z 11.900} C_DIS
   LIN {X -10.616, Y -15.823, Z 11.900} C_DIS
   LIN {X -11.366, Y -17.081, Z 11.900} C_DIS
   LIN {X -12.243, Y -18.567, Z 11.900} C_DIS
   LIN {X -12.741, Y -19.825, Z 11.900} C_DIS
   LIN {X -13.422, Y -21.510, Z 11.900} C_DIS
   LIN {X -13.481, Y -23.132, Z 11.900} C_DIS
   LIN {X -13.496, Y -24.750, Z 11.900} C_DIS
   LIN {X -12.890, Y -26.528, Z 11.900} C_DIS
   LIN {X -12.572, Y -27.539, Z 11.900} C_DIS
   LIN {X -12.096, Y -28.189, Z 11.900} C_DIS
   LIN {X -11.283, Y -29.349, Z 11.900} C_DIS
   LIN {X -10.837, Y -29.829, Z 11.900} C_DIS
   LIN {X -9.873, Y -30.616, Z 11.900} C_DIS
   LIN {X -9.699, Y -30.747, Z 11.900} C_DIS
   LIN {X -9.462, Y -30.877, Z 11.900} C_DIS
   LIN {X -8.749, Y -31.269, Z 11.900} C_DIS
   LIN {X -7.786, Y -31.665, Z 11.900} C_DIS
   LIN {X -6.872, Y -31.991, Z 11.900} C_DIS
   LIN {X -5.590, Y -32.248, Z 11.900} C_DIS
   LIN {X -4.181, Y -32.192, Z 11.900} C_DIS
   LIN {X -2.535, Y -32.031, Z 11.900} C_DIS
   LIN {X -0.370, Y -31.166, Z 11.900} C_DIS
   LIN {X -0.062, Y -31.049, Z 11.900} C_DIS
   LIN {X 0.072, Y -30.942, Z 11.900} C_DIS
   LIN {X 2.163, Y -29.206, Z 11.900} C_DIS
   LIN {X 3.515, Y -26.830, Z 11.900} C_DIS
   LIN {X 4.001, Y -25.960, Z 11.900} C_DIS
   LIN {X 4.145, Y -25.480, Z 11.900} C_DIS
   LIN {X 4.569, Y -24.089, Z 11.900} C_DIS
   LIN {X 5.183, Y -21.932, Z 11.900} C_DIS
   LIN {X 5.372, Y -21.237, Z 11.900} C_DIS
   LIN {X 6.080, Y -18.371, Z 11.900} C_DIS
   LIN {X 6.358, Y -17.254, Z 11.900} C_DIS
   LIN {X 6.410, Y -17.030, Z 11.900} C_DIS
   LIN {X 7.326, Y -12.488, Z 11.900} C_DIS
   LIN {X 7.671, Y -10.477, Z 11.900} C_DIS
   LIN {X 8.043, Y -8.071, Z 11.900} C_DIS
   LIN {X 8.384, Y -5.405, Z 11.900} C_DIS
   LIN {X 8.483, Y -4.496, Z 11.900} C_DIS
   LIN {X 8.568, Y -3.531, Z 11.900} C_DIS
   LIN {X 8.746, Y -1.671, Z 11.900} C_DIS
   LIN {X 8.873, Y -0.004, Z 11.900} C_DIS
   LIN {X 8.973, Y 1.704, Z 11.900} C_DIS
   LIN {X 9.030, Y 2.901, Z 11.900} C_DIS
   LIN {X 9.060, Y 3.981, Z 11.900} C_DIS
   LIN {X 9.110, Y 6.206, Z 11.900} C_DIS
   LIN {X 9.104, Y 7.826, Z 11.900} C_DIS
   LIN {X 9.100, Y 8.992, Z 11.900} C_DIS
   LIN {X 9.053, Y 10.747, Z 11.900} C_DIS
   LIN {X 8.989, Y 12.467, Z 11.900} C_DIS
   LIN {X 8.886, Y 14.247, Z 11.900} C_DIS
   LIN {X 8.776, Y 15.761, Z 11.900} C_DIS
   LIN {X 8.523, Y 18.615, Z 11.900} C_DIS
   LIN {X 8.421, Y 19.490, Z 11.900} C_DIS
   LIN {X 8.001, Y 22.811, Z 11.900} C_DIS
   LIN {X 7.859, Y 23.812, Z 11.900} C_DIS
   LIN {X 7.751, Y 24.463, Z 11.900} C_DIS
   LIN {X 7.477, Y 26.172, Z 11.900} C_DIS
   LIN {X 7.111, Y 28.054, Z 11.900} C_DIS
   LIN {X 6.571, Y 30.811, Z 11.900} C_DIS
   LIN {X 6.123, Y 32.749, Z 11.900} C_DIS
   LIN {X 6.039, Y 33.118, Z 11.900} C_DIS
   LIN {X 5.376, Y 35.731, Z 11.900}
   LaserEnd_Ext()
   LIN {X 2.144, Y 40.522, Z 11.900}
   LaserStart_Ext()
   LIN {X -1.105, Y 40.522, Z 11.900}
   LaserEnd_Ext()
   LIN {X -1.998, Y 39.522, Z 11.900}
   LaserStart_Ext()
   LIN {X 3.103, Y 39.522, Z 11.900}
   LaserEnd_Ext()
   LIN {X 3.551, Y 38.522, Z 11.900}
   LaserStart_Ext()
   LIN {X -2.361, Y 38.522, Z 11.900}
   LaserEnd_Ext()
   LIN {X -2.313, Y 37.522, Z 11.900}
   LaserStart_Ext()
   LIN {X 3.844, Y 37.522, Z 11.900}
   LaserEnd_Ext()
   LIN {X 4.122, Y 36.522, Z 11.900}
   LaserStart_Ext()
   LIN {X -2.131, Y 36.522, Z 11.900}
   LaserEnd_Ext()
   LIN {X -1.914, Y 35.522, Z 11.900}
   LaserStart_Ext()
   LIN {X 4.398, Y 35.522, Z 11.900}
   LaserEnd_Ext()
   LIN {X 4.651, Y 34.522, Z 11.900}
   LaserStart_Ext()
   LIN {X -1.701, Y 34.522, Z 11.900}
   LaserEnd_Ext()
   LIN {X -1.516, Y 33.522, Z 11.900}
   LaserStart_Ext()
   LIN {X 4.905, Y 33.522, Z 11.900}
   LaserEnd_Ext()
   LIN {X 5.149, Y 32.522, Z 11.900}
   LaserStart_Ext()
   LIN {X -1.332, Y 32.522, Z 11.900}
   LaserEnd_Ext()
   LIN {X -1.173, Y 31.522, Z 11.900}
   LaserStart_Ext()
   LIN {X 5.380, Y 31.522, Z 11.900}
   LaserEnd_Ext()
   LIN {X 5.608, Y 30.522, Z 11.900}
   LaserStart_Ext()
   LIN {X -1.025, Y 30.522, Z 11.900}
   LaserEnd_Ext()
   LIN {X -0.877, Y 29.522, Z 11.900}
   LaserStart_Ext()
   LIN {X 5.804, Y 29.522, Z 11.900}
   LaserEnd_Ext()
   LIN {X 6.001, Y 28.522, Z 11.900}
   LaserStart_Ext()
   LIN {X -0.764, Y 28.522, Z 11.900}
   LaserEnd_Ext()
   LIN {X -0.662, Y 27.522, Z 11.900}
   LaserStart_Ext()
   LIN {X 6.196, Y 27.522, Z 11.900}
   LaserEnd_Ext()
   LIN {X 6.391, Y 26.522, Z 11.900}
   LaserStart_Ext()
   LIN {X -0.552, Y 26.522, Z 11.900}
   LaserEnd_Ext()
   LIN {X -0.468, Y 25.522, Z 11.900}
   LaserStart_Ext()
   LIN {X 6.569, Y 25.522, Z 11.900}
   LaserEnd_Ext()
   LIN {X 6.729, Y 24.522, Z 11.900}
   LaserStart_Ext()
   LIN {X -0.410, Y 24.522, Z 11.900}
   LaserEnd_Ext()
   LIN {X -0.344, Y 23.522, Z 11.900}
   LaserStart_Ext()
   LIN {X 6.890, Y 23.522, Z 11.900}
   LaserEnd_Ext()
   LIN {X 7.029, Y 22.522, Z 11.900}
   LaserStart_Ext()
   LIN {X -0.300, Y 22.522, Z 11.900}
   LaserEnd_Ext()
   LIN {X -0.275, Y 21.522, Z 11.900}
   LaserStart_Ext()
   LIN {X 7.156, Y 21.522, Z 11.900}
   LaserEnd_Ext()
   LIN {X 7.282, Y 20.522, Z 11.900}
   LaserStart_Ext()
   LIN {X -0.264, Y 20.522, Z 11.900}
   LaserEnd_Ext()
   LIN {X -0.265, Y 19.522, Z 11.900}
   LaserStart_Ext()
   LIN {X 7.409, Y 19.522, Z 11.900}
   LaserEnd_Ext()
   LIN {X 7.527, Y 18.522, Z 11.900}
   LaserStart_Ext()
   LIN {X -0.267, Y 18.522, Z 11.900}
   LaserEnd_Ext()
   LIN {X -0.285, Y 17.522, Z 11.900}
   LaserStart_Ext()
   LIN {X 7.616, Y 17.522, Z 11.900}
   LaserEnd_Ext()
   LIN {X 7.705, Y 16.522, Z 11.900}
   LaserStart_Ext()
   LIN {X -0.326, Y 16.522, Z 11.900}
   LaserEnd_Ext()
   LIN {X -0.381, Y 15.522, Z 11.900}
   LaserStart_Ext()
   LIN {X 7.791, Y 15.522, Z 11.900}
   LaserEnd_Ext()
   LIN {X 7.864, Y 14.522, Z 11.900}
   LaserStart_Ext()
   LIN {X -0.459, Y 14.522, Z 11.900}
   LaserEnd_Ext()
   LIN {X -0.538, Y 13.522, Z 11.900}
   LaserStart_Ext()
   LIN {X 7.927, Y 13.522, Z 11.900}
   LaserEnd_Ext()
   LIN {X 7.985, Y 12.522, Z 11.900}
   LaserStart_Ext()
   LIN {X -0.620, Y 12.522, Z 11.900}
   LaserEnd_Ext()
   LIN {X -0.731, Y 11.522, Z 11.900}
   LaserStart_Ext()
   LIN {X 8.024, Y 11.522, Z 11.900}
   LaserEnd_Ext()
   LIN {X 8.059, Y 10.522, Z 11.900}
   LaserStart_Ext()
   LIN {X -0.858, Y 10.522, Z 11.900}
   LaserEnd_Ext()
   LIN {X -0.993, Y 9.522, Z 11.900}
   LaserStart_Ext()
   LIN {X 8.086, Y 9.522, Z 11.900}
   LaserEnd_Ext()
   LIN {X 8.102, Y 8.522, Z 11.900}
   LaserStart_Ext()
   LIN {X -1.141, Y 8.522, Z 11.900}
   LaserEnd_Ext()
   LIN {X -1.298, Y 7.522, Z 11.900}
   LaserStart_Ext()
   LIN {X 8.105, Y 7.522, Z 11.900}
   LaserEnd_Ext()
   LIN {X 8.109, Y 6.522, Z 11.900}
   LaserStart_Ext()
   LIN {X -1.465, Y 6.522, Z 11.900}
   LaserEnd_Ext()
   LIN {X -1.686, Y 5.522, Z 11.900}
   LaserStart_Ext()
   LIN {X 8.094, Y 5.522, Z 11.900}
   LaserEnd_Ext()
   LIN {X 8.072, Y 4.522, Z 11.900}
   LaserStart_Ext()
   LIN {X -1.906, Y 4.522, Z 11.900}
   LaserEnd_Ext()
   LIN {X -2.127, Y 3.522, Z 11.900}
   LaserStart_Ext()
   LIN {X 8.047, Y 3.522, Z 11.900}
   LaserEnd_Ext()
   LIN {X 8.011, Y 2.522, Z 11.900}
   LaserStart_Ext()
   LIN {X -2.338, Y 2.522, Z 11.900}
   LaserEnd_Ext()
   LIN {X -2.571, Y 1.522, Z 11.900}
   LaserStart_Ext()
   LIN {X 7.961, Y 1.522, Z 11.900}
   LaserEnd_Ext()
   LIN {X 7.902, Y 0.522, Z 11.900}
   LaserStart_Ext()
   LIN {X -2.864, Y 0.522, Z 11.900}
   LaserEnd_Ext()
   LIN {X -3.178, Y -0.478, Z 11.900}
   LaserStart_Ext()
   LIN {X 7.834, Y -0.478, Z 11.900}
   LaserEnd_Ext()
   LIN {X 7.758, Y -1.478, Z 11.900}
   LaserStart_Ext()
   LIN {X -3.475, Y -1.478, Z 11.900}
   LaserEnd_Ext()
   LIN {X -3.773, Y -2.478, Z 11.900}
   LaserStart_Ext()
   LIN {X 7.664, Y -2.478, Z 11.900}
   LaserEnd_Ext()
   LIN {X 7.569, Y -3.478, Z 11.900}
   LaserStart_Ext()
   LIN {X -4.070, Y -3.478, Z 11.900}
   LaserEnd_Ext()
   LIN {X -4.407, Y -4.478, Z 11.900}
   LaserStart_Ext()
   LIN {X 7.479, Y -4.478, Z 11.900}
   LaserEnd_Ext()
   LIN {X 7.366, Y -5.478, Z 11.900}
   LaserStart_Ext()
   LIN {X -4.786, Y -5.478, Z 11.900}
   LaserEnd_Ext()
   LIN {X -5.168, Y -6.478, Z 11.900}
   LaserStart_Ext()
   LIN {X 7.239, Y -6.478, Z 11.900}
   LaserEnd_Ext()
   LIN {X 7.111, Y -7.478, Z 11.900}
   LaserStart_Ext()
   LIN {X -5.551, Y -7.478, Z 11.900}
   LaserEnd_Ext()
   LIN {X -5.934, Y -8.478, Z 11.900}
   LaserStart_Ext()
   LIN {X 6.968, Y -8.478, Z 11.900}
   LaserEnd_Ext()
   LIN {X 6.814, Y -9.478, Z 11.900}
   LaserStart_Ext()
   LIN {X -6.369, Y -9.478, Z 11.900}
   LaserEnd_Ext()
   LIN {X -6.817, Y -10.478, Z 11.900}
   LaserStart_Ext()
   LIN {X 6.656, Y -10.478, Z 11.900}
   LaserEnd_Ext()
   LIN {X 6.484, Y -11.478, Z 11.900}
   LaserStart_Ext()
   LIN {X -7.269, Y -11.478, Z 11.900}
   LaserEnd_Ext()
   LIN {X -7.736, Y -12.478, Z 11.900}
   LaserStart_Ext()
   LIN {X 6.307, Y -12.478, Z 11.900}
   LaserEnd_Ext()
   LIN {X 6.106, Y -13.478, Z 11.900}
   LaserStart_Ext()
   LIN {X -8.249, Y -13.478, Z 11.900}
   LaserEnd_Ext()
   LIN {X -8.776, Y -14.478, Z 11.900}
   LaserStart_Ext()
   LIN {X 5.904, Y -14.478, Z 11.900}
   LaserEnd_Ext()
   LIN {X 5.702, Y -15.478, Z 11.900}
   LaserStart_Ext()
   LIN {X -9.304, Y -15.478, Z 11.900}
   LaserEnd_Ext()
   LIN {X -9.843, Y -16.478, Z 11.900}
   LaserStart_Ext()
   LIN {X 5.501, Y -16.478, Z 11.900}
   LaserEnd_Ext()
   LIN {X 5.272, Y -17.478, Z 11.900}
   LaserStart_Ext()
   LIN {X -10.438, Y -17.478, Z 11.900}
   LaserEnd_Ext()
   LIN {X -11.029, Y -18.478, Z 11.900}
   LaserStart_Ext()
   LIN {X 5.023, Y -18.478, Z 11.900}
   LaserEnd_Ext()
   LIN {X 4.776, Y -19.478, Z 11.900}
   LaserStart_Ext()
   LIN {X -3.201, Y -19.478, Z 11.900}
   LaserEnd_Ext()
   LIN {X -5.784, Y -19.478, Z 11.900}
   LaserStart_Ext()
   LIN {X -11.528, Y -19.478, Z 11.900}
   LaserEnd_Ext()
   LIN {X -11.927, Y -20.478, Z 11.900}
   LaserStart_Ext()
   LIN {X -7.343, Y -20.478, Z 11.900}
   LaserEnd_Ext()
   LIN {X -1.884, Y -20.478, Z 11.900}
   LaserStart_Ext()
   LIN {X 4.529, Y -20.478, Z 11.900}
   LaserEnd_Ext()
   LIN {X 4.270, Y -21.478, Z 11.900}
   LaserStart_Ext()
   LIN {X -1.077, Y -21.478, Z 11.900}
   LaserEnd_Ext()
   LIN {X -8.059, Y -21.478, Z 11.900}
   LaserStart_Ext()
   LIN {X -12.331, Y -21.478, Z 11.900}
   LaserEnd_Ext()
   LIN {X -12.456, Y -22.478, Z 11.900}
   LaserStart_Ext()
   LIN {X -8.330, Y -22.478, Z 11.900}
   LaserEnd_Ext()
   LIN {X -0.768, Y -22.478, Z 11.900}
   LaserStart_Ext()
   LIN {X 3.988, Y -22.478, Z 11.900}
   LaserEnd_Ext()
   LIN {X 3.703, Y -23.478, Z 11.900}
   LaserStart_Ext()
   LIN {X -0.784, Y -23.478, Z 11.900}
   LaserEnd_Ext()
   LIN {X -8.409, Y -23.478, Z 11.900}
   LaserStart_Ext()
   LIN {X -12.484, Y -23.478, Z 11.900}
   LaserEnd_Ext()
   LIN {X -12.494, Y -24.478, Z 11.900}
   LaserStart_Ext()
   LIN {X -8.061, Y -24.478, Z 11.900}
   LaserEnd_Ext()
   LIN {X -0.996, Y -24.478, Z 11.900}
   LaserStart_Ext()
   LIN {X 3.405, Y -24.478, Z 11.900}
   LaserEnd_Ext()
   LIN {X 3.102, Y -25.478, Z 11.900}
   LaserStart_Ext()
   LIN {X -1.674, Y -25.478, Z 11.900}
   LaserEnd_Ext()
   LIN {X -7.638, Y -25.478, Z 11.900}
   LaserStart_Ext()
   LIN {X -12.191, Y -25.478, Z 11.900}
   LaserEnd_Ext()
   LIN {X -11.857, Y -26.478, Z 11.900}
   LaserStart_Ext()
   LIN {X -6.469, Y -26.478, Z 11.900}
   LaserEnd_Ext()
   LIN {X -2.666, Y -26.478, Z 11.900}
   LaserStart_Ext()
   LIN {X 2.565, Y -26.478, Z 11.900}
   LaserEnd_Ext()
   LIN {X 1.996, Y -27.478, Z 11.900}
   LaserStart_Ext()
   LIN {X -11.377, Y -27.478, Z 11.900}
   LaserEnd_Ext()
   LIN {X -10.672, Y -28.478, Z 11.900}
   LaserStart_Ext()
   LIN {X 1.427, Y -28.478, Z 11.900}
   LaserEnd_Ext()
   LIN {X 0.269, Y -29.478, Z 11.900}
   LaserStart_Ext()
   LIN {X -9.685, Y -29.478, Z 11.900}
   LaserEnd_Ext()
   LIN {X -8.042, Y -30.478, Z 11.900}
   LaserStart_Ext()
   LIN {X -1.344, Y -30.478, Z 11.900}
   LaserEnd_Ext()
   LIN {X -3.075, Y -19.551, Z 12.750}
   LaserStart_Ext()
   LIN {X -4.112, Y -19.254, Z 12.750} C_DIS
   LIN {X -4.898, Y -19.398, Z 12.750} C_DIS
   LIN {X -5.566, Y -19.452, Z 12.750} C_DIS
   LIN {X -6.432, Y -19.847, Z 12.750} C_DIS
   LIN {X -7.078, Y -20.379, Z 12.750} C_DIS
   LIN {X -7.796, Y -21.370, Z 12.750} C_DIS
   LIN {X -8.031, Y -21.981, Z 12.750} C_DIS
   LIN {X -8.177, Y -23.359, Z 12.750} C_DIS
   LIN {X -8.148, Y -23.616, Z 12.750} C_DIS
   LIN {X -8.036, Y -23.929, Z 12.750} C_DIS
   LIN {X -7.670, Y -24.935, Z 12.750} C_DIS
   LIN {X -7.348, Y -25.364, Z 12.750} C_DIS
   LIN {X -7.191, Y -25.580, Z 12.750} C_DIS
   LIN {X -6.785, Y -25.924, Z 12.750} C_DIS
   LIN {X -6.583, Y -26.097, Z 12.750} C_DIS
   LIN {X -6.100, Y -26.375, Z 12.750} C_DIS
   LIN {X -5.325, Y -26.634, Z 12.750} C_DIS
   LIN {X -5.196, Y -26.673, Z 12.750} C_DIS
   LIN {X -4.404, Y -26.718, Z 12.750} C_DIS
   LIN {X -4.211, Y -26.727, Z 12.750} C_DIS
   LIN {X -3.910, Y -26.684, Z 12.750} C_DIS
   LIN {X -3.278, Y -26.527, Z 12.750} C_DIS
   LIN {X -2.758, Y -26.308, Z 12.750} C_DIS
   LIN {X -2.495, Y -26.164, Z 12.750} C_DIS
   LIN {X -2.307, Y -26.037, Z 12.750} C_DIS
   LIN {X -0.994, Y -24.003, Z 12.750} C_DIS
   LIN {X -0.824, Y -23.790, Z 12.750} C_DIS
   LIN {X -0.769, Y -23.474, Z 12.750} C_DIS
   LIN {X -0.857, Y -22.635, Z 12.750} C_DIS
   LIN {X -0.920, Y -21.746, Z 12.750} C_DIS
   LIN {X -1.082, Y -21.396, Z 12.750} C_DIS
   LIN {X -1.346, Y -20.903, Z 12.750} C_DIS
   LIN {X -2.504, Y -19.831, Z 12.750} C_DIS
   LIN {X -2.753, Y -19.640, Z 12.750} C_DIS
   LIN {X -3.075, Y -19.551, Z 12.750}
   LaserEnd_Ext()
   LIN {X 4.417, Y -24.771, Z 12.750}
   LaserStart_Ext()
   LIN {X 4.645, Y -24.022, Z 12.750} C_DIS
   LIN {X 4.976, Y -22.862, Z 12.750} C_DIS
   LIN {X 5.527, Y -20.830, Z 12.750} C_DIS
   LIN {X 6.251, Y -17.898, Z 12.750} C_DIS
   LIN {X 6.452, Y -17.028, Z 12.750} C_DIS
   LIN {X 7.270, Y -12.913, Z 12.750} C_DIS
   LIN {X 7.453, Y -12.006, Z 12.750} C_DIS
   LIN {X 7.508, Y -11.690, Z 12.750} C_DIS
   LIN {X 8.096, Y -7.887, Z 12.750} C_DIS
   LIN {X 8.320, Y -6.135, Z 12.750} C_DIS
   LIN {X 8.551, Y -4.020, Z 12.750} C_DIS
   LIN {X 8.749, Y -1.773, Z 12.750} C_DIS
   LIN {X 8.803, Y -1.208, Z 12.750} C_DIS
   LIN {X 8.842, Y -0.701, Z 12.750} C_DIS
   LIN {X 8.994, Y 1.906, Z 12.750} C_DIS
   LIN {X 9.032, Y 2.693, Z 12.750} C_DIS
   LIN {X 9.078, Y 4.343, Z 12.750} C_DIS
   LIN {X 9.110, Y 5.815, Z 12.750} C_DIS
   LIN {X 9.102, Y 8.319, Z 12.750} C_DIS
   LIN {X 9.099, Y 9.027, Z 12.750} C_DIS
   LIN {X 9.070, Y 10.094, Z 12.750} C_DIS
   LIN {X 8.982, Y 12.502, Z 12.750} C_DIS
   LIN {X 8.918, Y 13.602, Z 12.750} C_DIS
   LIN {X 8.732, Y 16.151, Z 12.750} C_DIS
   LIN {X 8.552, Y 18.188, Z 12.750} C_DIS
   LIN {X 8.479, Y 18.813, Z 12.750} C_DIS
   LIN {X 7.905, Y 23.343, Z 12.750} C_DIS
   LIN {X 7.487, Y 25.959, Z 12.750} C_DIS
   LIN {X 6.930, Y 28.825, Z 12.750} C_DIS
   LIN {X 6.591, Y 30.553, Z 12.750} C_DIS
   LIN {X 6.012, Y 33.061, Z 12.750} C_DIS
   LIN {X 5.827, Y 33.798, Z 12.750} C_DIS
   LIN {X 5.290, Y 35.891, Z 12.750} C_DIS
   LIN {X 4.824, Y 37.567, Z 12.750} C_DIS
   LIN {X 4.767, Y 37.767, Z 12.750} C_DIS
   LIN {X 4.696, Y 38.007, Z 12.750} C_DIS
   LIN {X 4.325, Y 39.262, Z 12.750} C_DIS
   LIN {X 3.881, Y 40.124, Z 12.750} C_DIS
   LIN {X 3.648, Y 40.572, Z 12.750} C_DIS
   LIN {X 2.882, Y 41.206, Z 12.750} C_DIS
   LIN {X 2.306, Y 41.685, Z 12.750} C_DIS
   LIN {X 1.933, Y 41.782, Z 12.750} C_DIS
   LIN {X 0.613, Y 42.124, Z 12.750} C_DIS
   LIN {X -0.912, Y 41.628, Z 12.750} C_DIS
   LIN {X -1.845, Y 41.365, Z 12.750} C_DIS
   LIN {X -2.406, Y 40.794, Z 12.750} C_DIS
   LIN {X -2.903, Y 40.221, Z 12.750} C_DIS
   LIN {X -3.162, Y 39.394, Z 12.750} C_DIS
   LIN {X -3.460, Y 38.581, Z 12.750} C_DIS
   LIN {X -3.381, Y 37.401, Z 12.750} C_DIS
   LIN {X -3.363, Y 37.194, Z 12.750} C_DIS
   LIN {X -3.330, Y 37.053, Z 12.750} C_DIS
   LIN {X -3.084, Y 35.974, Z 12.750} C_DIS
   LIN {X -2.807, Y 34.693, Z 12.750} C_DIS
   LIN {X -2.747, Y 34.410, Z 12.750} C_DIS
   LIN {X -2.658, Y 33.930, Z 12.750} C_DIS
   LIN {X -2.311, Y 32.078, Z 12.750} C_DIS
   LIN {X -2.051, Y 30.354, Z 12.750} C_DIS
   LIN {X -1.882, Y 29.214, Z 12.750} C_DIS
   LIN {X -1.843, Y 28.834, Z 12.750} C_DIS
   LIN {X -1.752, Y 27.948, Z 12.750} C_DIS
   LIN {X -1.523, Y 25.881, Z 12.750} C_DIS
   LIN {X -1.369, Y 23.183, Z 12.750} C_DIS
   LIN {X -1.344, Y 22.833, Z 12.750} C_DIS
   LIN {X -1.324, Y 22.490, Z 12.750} C_DIS
   LIN {X -1.297, Y 21.386, Z 12.750} C_DIS
   LIN {X -1.302, Y 17.905, Z 12.750} C_DIS
   LIN {X -1.306, Y 17.567, Z 12.750} C_DIS
   LIN {X -1.315, Y 17.287, Z 12.750} C_DIS
   LIN {X -1.325, Y 17.063, Z 12.750} C_DIS
   LIN {X -1.383, Y 15.732, Z 12.750} C_DIS
   LIN {X -1.484, Y 14.447, Z 12.750} C_DIS
   LIN {X -1.680, Y 12.063, Z 12.750} C_DIS
   LIN {X -1.869, Y 10.581, Z 12.750} C_DIS
   LIN {X -2.342, Y 7.390, Z 12.750} C_DIS
   LIN {X -2.479, Y 6.569, Z 12.750} C_DIS
   LIN {X -3.503, Y 1.929, Z 12.750} C_DIS
   LIN {X -3.526, Y 1.818, Z 12.750} C_DIS
   LIN {X -3.552, Y 1.709, Z 12.750} C_DIS
   LIN {X -3.617, Y 1.498, Z 12.750} C_DIS
   LIN {X -5.129, Y -3.585, Z 12.750} C_DIS
   LIN {X -5.469, Y -4.483, Z 12.750} C_DIS
   LIN {X -7.084, Y -8.702, Z 12.750} C_DIS
   LIN {X -7.794, Y -10.286, Z 12.750} C_DIS
   LIN {X -8.853, Y -12.554, Z 12.750} C_DIS
   LIN {X -10.496, Y -15.671, Z 12.750} C_DIS
   LIN {X -10.564, Y -15.799, Z 12.750} C_DIS
   LIN {X -10.662, Y -15.969, Z 12.750} C_DIS
   LIN {X -12.181, Y -18.540, Z 12.750} C_DIS
   LIN {X -13.181, Y -21.064, Z 12.750} C_DIS
   LIN {X -13.352, Y -21.487, Z 12.750} C_DIS
   LIN {X -13.367, Y -21.894, Z 12.750} C_DIS
   LIN {X -13.395, Y -24.859, Z 12.750} C_DIS
   LIN {X -12.575, Y -27.267, Z 12.750} C_DIS
   LIN {X -12.459, Y -27.567, Z 12.750} C_DIS
   LIN {X -12.265, Y -27.861, Z 12.750} C_DIS
   LIN {X -11.411, Y -29.078, Z 12.750} C_DIS
   LIN {X -10.700, Y -29.845, Z 12.750} C_DIS
   LIN {X -10.411, Y -30.081, Z 12.750} C_DIS
   LIN {X -9.370, Y -30.866, Z 12.750} C_DIS
   LIN {X -8.489, Y -31.351, Z 12.750} C_DIS
   LIN {X -7.795, Y -31.645, Z 12.750} C_DIS
   LIN {X -7.199, Y -31.857, Z 12.750} C_DIS
   LIN {X -5.410, Y -32.216, Z 12.750} C_DIS
   LIN {X -5.213, Y -32.208, Z 12.750} C_DIS
   LIN {X -2.195, Y -31.913, Z 12.750} C_DIS
   LIN {X -0.458, Y -31.220, Z 12.750} C_DIS
   LIN {X 0.074, Y -30.966, Z 12.750} C_DIS
   LIN {X 1.022, Y -30.166, Z 12.750} C_DIS
   LIN {X 2.251, Y -29.147, Z 12.750} C_DIS
   LIN {X 2.944, Y -27.928, Z 12.750} C_DIS
   LIN {X 4.081, Y -25.895, Z 12.750} C_DIS
   LIN {X 4.417, Y -24.771, Z 12.750}
   LaserEnd_Ext()
   LIN {X -12.280, Y -21.503, Z 12.750}
   LaserStart_Ext()
   LIN {X -12.280, Y -25.032, Z 12.750}
   LaserEnd_Ext()
   LIN {X -11.280, Y -27.524, Z 12.750}
   LaserStart_Ext()
   LIN {X -11.280, Y -18.981, Z 12.750}
   LaserEnd_Ext()
   LIN {X -10.280, Y -17.288, Z 12.750}
   LaserStart_Ext()
   LIN {X -10.280, Y -28.827, Z 12.750}
   LaserEnd_Ext()
   LIN {X -9.280, Y -29.681, Z 12.750}
   LaserStart_Ext()
   LIN {X -9.280, Y -15.509, Z 12.750}
   LaserEnd_Ext()
   LIN {X -8.280, Y -13.611, Z 12.750}
   LaserStart_Ext()
   LIN {X -8.280, Y -20.334, Z 12.750}
   LaserEnd_Ext()
   LIN {X -8.280, Y -25.788, Z 12.750}
   LaserStart_Ext()
   LIN {X -8.280, Y -30.325, Z 12.750}
   LaserEnd_Ext()
   LIN {X -7.280, Y -30.767, Z 12.750}
   LaserStart_Ext()
   LIN {X -7.280, Y -26.817, Z 12.750}
   LaserEnd_Ext()
   LIN {X -7.280, Y -19.250, Z 12.750}
   LaserStart_Ext()
   LIN {X -7.280, Y -11.549, Z 12.750}
   LaserEnd_Ext()
   LIN {X -6.280, Y -9.354, Z 12.750}
   LaserStart_Ext()
   LIN {X -6.280, Y -18.678, Z 12.750}
   LaserEnd_Ext()
   LIN {X -6.280, Y -27.369, Z 12.750}
   LaserStart_Ext()
   LIN {X -6.280, Y -31.022, Z 12.750}
   LaserEnd_Ext()
   LIN {X -5.280, Y -31.210, Z 12.750}
   LaserStart_Ext()
   LIN {X -5.280, Y -27.669, Z 12.750}
   LaserEnd_Ext()
   LIN {X -5.280, Y -18.425, Z 12.750}
   LaserStart_Ext()
   LIN {X -5.280, Y -6.787, Z 12.750}
   LaserEnd_Ext()
   LIN {X -4.280, Y -4.168, Z 12.750}
   LaserStart_Ext()
   LIN {X -4.280, Y -18.269, Z 12.750}
   LaserEnd_Ext()
   LIN {X -4.280, Y -27.725, Z 12.750}
   LaserStart_Ext()
   LIN {X -4.280, Y -31.112, Z 12.750}
   LaserEnd_Ext()
   LIN {X -3.280, Y -31.015, Z 12.750}
   LaserStart_Ext()
   LIN {X -3.280, Y -27.558, Z 12.750}
   LaserEnd_Ext()
   LIN {X -3.280, Y -18.452, Z 12.750}
   LaserStart_Ext()
   LIN {X -3.280, Y -0.877, Z 12.750}
   LaserEnd_Ext()
   LIN {X -2.280, Y 38.894, Z 12.750}
   LaserStart_Ext()
   LIN {X -2.280, Y 36.945, Z 12.750}
   LaserEnd_Ext()
   LIN {X -2.280, Y 2.832, Z 12.750}
   LaserStart_Ext()
   LIN {X -2.280, Y -18.760, Z 12.750}
   LaserEnd_Ext()
   LIN {X -2.280, Y -27.186, Z 12.750}
   LaserStart_Ext()
   LIN {X -2.280, Y -30.871, Z 12.750}
   LaserEnd_Ext()
   LIN {X -1.280, Y -30.471, Z 12.750}
   LaserStart_Ext()
   LIN {X -1.280, Y -26.290, Z 12.750}
   LaserEnd_Ext()
   LIN {X -1.280, Y -19.602, Z 12.750}
   LaserStart_Ext()
   LIN {X -1.280, Y 7.737, Z 12.750}
   LaserEnd_Ext()
   LIN {X -1.280, Y 31.947, Z 12.750}
   LaserStart_Ext()
   LIN {X -1.280, Y 40.486, Z 12.750}
   LaserEnd_Ext()
   LIN {X -0.280, Y 40.782, Z 12.750}
   LaserStart_Ext()
   LIN {X -0.280, Y -20.776, Z 12.750}
   LaserEnd_Ext()
   LIN {X -0.280, Y -24.741, Z 12.750}
   LaserStart_Ext()
   LIN {X -0.280, Y -29.956, Z 12.750}
   LaserEnd_Ext()
   LIN {X 0.720, Y -29.118, Z 12.750}
   LaserStart_Ext()
   LIN {X 0.720, Y 41.063, Z 12.750}
   LaserEnd_Ext()
   LIN {X 1.720, Y 40.805, Z 12.750}
   LaserStart_Ext()
   LIN {X 1.720, Y -28.058, Z 12.750}
   LaserEnd_Ext()
   LIN {X 2.720, Y -26.279, Z 12.750}
   LaserStart_Ext()
   LIN {X 2.720, Y 40.042, Z 12.750}
   LaserEnd_Ext()
   LIN {X 3.720, Y 37.780, Z 12.750}
   LaserStart_Ext()
   LIN {X 3.720, Y -23.620, Z 12.750}
   LaserEnd_Ext()
   LIN {X 4.720, Y -19.925, Z 12.750}
   LaserStart_Ext()
   LIN {X 4.720, Y 34.089, Z 12.750}
   LaserEnd_Ext()
   LIN {X 5.720, Y 29.796, Z 12.750}
   LaserStart_Ext()
   LIN {X 5.720, Y -15.582, Z 12.750}
   LaserEnd_Ext()
   LIN {X 6.720, Y -10.240, Z 12.750}
   LaserStart_Ext()
   LIN {X 6.720, Y 24.425, Z 12.750}
   LaserEnd_Ext()
   LIN {X 7.720, Y 16.246, Z 12.750}
   LaserStart_Ext()
   LIN {X 7.720, Y -2.055, Z 12.750}
   LaserEnd_Ext()
   LIN {X -3.512, Y -27.394, Z 13.600}
   LaserStart_Ext()
   LIN {X -3.016, Y -27.272, Z 13.600} C_DIS
   LIN {X -2.334, Y -26.988, Z 13.600} C_DIS
   LIN {X -1.796, Y -26.673, Z 13.600} C_DIS
   LIN {X -1.588, Y -26.532, Z 13.600} C_DIS
   LIN {X -1.048, Y -25.696, Z 13.600} C_DIS
   LIN {X -0.099, Y -24.502, Z 13.600} C_DIS
   LIN {X 0.211, Y -22.732, Z 13.600} C_DIS
   LIN {X 0.160, Y -22.250, Z 13.600} C_DIS
   LIN {X -0.079, Y -21.194, Z 13.600} C_DIS
   LIN {X -0.814, Y -19.994, Z 13.600} C_DIS
   LIN {X -0.887, Y -19.858, Z 13.600} C_DIS
   LIN {X -1.019, Y -19.736, Z 13.600} C_DIS
   LIN {X -2.282, Y -18.766, Z 13.600} C_DIS
   LIN {X -3.915, Y -18.316, Z 13.600} C_DIS
   LIN {X -6.108, Y -18.680, Z 13.600} C_DIS
   LIN {X -6.335, Y -18.746, Z 13.600} C_DIS
   LIN {X -8.001, Y -20.119, Z 13.600} C_DIS
   LIN {X -8.181, Y -20.367, Z 13.600} C_DIS
   LIN {X -8.892, Y -22.216, Z 13.600} C_DIS
   LIN {X -8.943, Y -22.698, Z 13.600} C_DIS
   LIN {X -8.774, Y -24.184, Z 13.600} C_DIS
   LIN {X -8.545, Y -24.822, Z 13.600} C_DIS
   LIN {X -8.251, Y -25.372, Z 13.600} C_DIS
   LIN {X -7.744, Y -26.047, Z 13.600} C_DIS
   LIN {X -7.058, Y -26.643, Z 13.600} C_DIS
   LIN {X -6.688, Y -26.883, Z 13.600} C_DIS
   LIN {X -6.478, Y -26.997, Z 13.600} C_DIS
   LIN {X -6.375, Y -27.050, Z 13.600} C_DIS
   LIN {X -6.256, Y -27.102, Z 13.600} C_DIS
   LIN {X -6.068, Y -27.182, Z 13.600} C_DIS
   LIN {X -5.678, Y -27.316, Z 13.600} C_DIS
   LIN {X -5.267, Y -27.411, Z 13.600} C_DIS
   LIN {X -5.035, Y -27.453, Z 13.600} C_DIS
   LIN {X -4.426, Y -27.491, Z 13.600} C_DIS
   LIN {X -4.266, Y -27.491, Z 13.600} C_DIS
   LIN {X -3.512, Y -27.394, Z 13.600}
   LaserEnd_Ext()
   LIN {X 8.537, Y 18.137, Z 13.600}
   LaserStart_Ext()
   LIN {X 8.193, Y 20.851, Z 13.600} C_DIS
   LIN {X 7.963, Y 22.790, Z 13.600} C_DIS
   LIN {X 7.756, Y 24.131, Z 13.600} C_DIS
   LIN {X 7.497, Y 25.746, Z 13.600} C_DIS
   LIN {X 6.748, Y 29.596, Z 13.600} C_DIS
   LIN {X 6.611, Y 30.296, Z 13.600} C_DIS
   LIN {X 6.300, Y 31.641, Z 13.600} C_DIS
   LIN {X 5.929, Y 33.245, Z 13.600} C_DIS
   LIN {X 5.358, Y 35.452, Z 13.600} C_DIS
   LIN {X 5.214, Y 36.013, Z 13.600} C_DIS
   LIN {X 5.145, Y 36.260, Z 13.600} C_DIS
   LIN {X 4.690, Y 37.873, Z 13.600} C_DIS
   LIN {X 4.359, Y 38.983, Z 13.600} C_DIS
   LIN {X 4.255, Y 39.328, Z 13.600} C_DIS
   LIN {X 4.018, Y 39.784, Z 13.600} C_DIS
   LIN {X 3.576, Y 40.636, Z 13.600} C_DIS
   LIN {X 3.017, Y 41.098, Z 13.600} C_DIS
   LIN {X 2.230, Y 41.746, Z 13.600} C_DIS
   LIN {X 0.777, Y 42.118, Z 13.600} C_DIS
   LIN {X 0.536, Y 42.180, Z 13.600} C_DIS
   LIN {X -0.154, Y 41.956, Z 13.600} C_DIS
   LIN {X -1.918, Y 41.405, Z 13.600} C_DIS
   LIN {X -2.028, Y 41.338, Z 13.600} C_DIS
   LIN {X -2.496, Y 40.779, Z 13.600} C_DIS
   LIN {X -3.052, Y 40.140, Z 13.600} C_DIS
   LIN {X -3.325, Y 39.265, Z 13.600} C_DIS
   LIN {X -3.539, Y 38.547, Z 13.600} C_DIS
   LIN {X -3.502, Y 38.096, Z 13.600} C_DIS
   LIN {X -3.428, Y 37.242, Z 13.600} C_DIS
   LIN {X -3.164, Y 36.100, Z 13.600} C_DIS
   LIN {X -3.132, Y 35.961, Z 13.600} C_DIS
   LIN {X -2.805, Y 34.458, Z 13.600} C_DIS
   LIN {X -2.456, Y 32.617, Z 13.600} C_DIS
   LIN {X -2.364, Y 32.128, Z 13.600} C_DIS
   LIN {X -2.238, Y 31.290, Z 13.600} C_DIS
   LIN {X -1.928, Y 29.265, Z 13.600} C_DIS
   LIN {X -1.852, Y 28.523, Z 13.600} C_DIS
   LIN {X -1.554, Y 25.824, Z 13.600} C_DIS
   LIN {X -1.352, Y 22.303, Z 13.600} C_DIS
   LIN {X -1.345, Y 22.199, Z 13.600} C_DIS
   LIN {X -1.339, Y 22.097, Z 13.600} C_DIS
   LIN {X -1.331, Y 21.767, Z 13.600} C_DIS
   LIN {X -1.338, Y 17.373, Z 13.600} C_DIS
   LIN {X -1.338, Y 17.273, Z 13.600} C_DIS
   LIN {X -1.414, Y 15.550, Z 13.600} C_DIS
   LIN {X -1.455, Y 15.015, Z 13.600} C_DIS
   LIN {X -1.713, Y 11.881, Z 13.600} C_DIS
   LIN {X -1.806, Y 11.159, Z 13.600} C_DIS
   LIN {X -2.478, Y 6.627, Z 13.600} C_DIS
   LIN {X -2.512, Y 6.423, Z 13.600} C_DIS
   LIN {X -2.812, Y 5.060, Z 13.600} C_DIS
   LIN {X -3.529, Y 1.788, Z 13.600} C_DIS
   LIN {X -4.522, Y -1.602, Z 13.600} C_DIS
   LIN {X -5.085, Y -3.496, Z 13.600} C_DIS
   LIN {X -5.194, Y -3.784, Z 13.600} C_DIS
   LIN {X -7.234, Y -9.112, Z 13.600} C_DIS
   LIN {X -7.505, Y -9.716, Z 13.600} C_DIS
   LIN {X -8.964, Y -12.839, Z 13.600} C_DIS
   LIN {X -10.034, Y -14.870, Z 13.600} C_DIS
   LIN {X -10.531, Y -15.809, Z 13.600} C_DIS
   LIN {X -11.258, Y -17.056, Z 13.600} C_DIS
   LIN {X -12.119, Y -18.513, Z 13.600} C_DIS
   LIN {X -12.893, Y -20.467, Z 13.600} C_DIS
   LIN {X -13.283, Y -21.462, Z 13.600} C_DIS
   LIN {X -13.271, Y -22.590, Z 13.600} C_DIS
   LIN {X -13.294, Y -24.969, Z 13.600} C_DIS
   LIN {X -12.798, Y -26.423, Z 13.600} C_DIS
   LIN {X -12.353, Y -27.582, Z 13.600} C_DIS
   LIN {X -11.604, Y -28.715, Z 13.600} C_DIS
   LIN {X -11.540, Y -28.807, Z 13.600} C_DIS
   LIN {X -11.437, Y -28.918, Z 13.600} C_DIS
   LIN {X -10.825, Y -29.597, Z 13.600} C_DIS
   LIN {X -10.437, Y -29.962, Z 13.600} C_DIS
   LIN {X -9.166, Y -30.902, Z 13.600} C_DIS
   LIN {X -8.971, Y -31.018, Z 13.600} C_DIS
   LIN {X -7.730, Y -31.591, Z 13.600} C_DIS
   LIN {X -7.029, Y -31.845, Z 13.600} C_DIS
   LIN {X -5.835, Y -32.086, Z 13.600} C_DIS
   LIN {X -5.232, Y -32.179, Z 13.600} C_DIS
   LIN {X -3.684, Y -31.975, Z 13.600} C_DIS
   LIN {X -1.854, Y -31.796, Z 13.600} C_DIS
   LIN {X -0.950, Y -31.435, Z 13.600} C_DIS
   LIN {X 0.210, Y -30.882, Z 13.600} C_DIS
   LIN {X 2.279, Y -29.137, Z 13.600} C_DIS
   LIN {X 2.373, Y -29.027, Z 13.600} C_DIS
   LIN {X 4.160, Y -25.829, Z 13.600} C_DIS
   LIN {X 4.689, Y -24.062, Z 13.600} C_DIS
   LIN {X 4.722, Y -23.956, Z 13.600} C_DIS
   LIN {X 4.768, Y -23.791, Z 13.600} C_DIS
   LIN {X 5.682, Y -20.422, Z 13.600} C_DIS
   LIN {X 6.080, Y -18.810, Z 13.600} C_DIS
   LIN {X 6.534, Y -16.849, Z 13.600} C_DIS
   LIN {X 7.319, Y -12.901, Z 13.600} C_DIS
   LIN {X 7.529, Y -11.768, Z 13.600} C_DIS
   LIN {X 7.815, Y -9.857, Z 13.600} C_DIS
   LIN {X 8.149, Y -7.703, Z 13.600} C_DIS
   LIN {X 8.256, Y -6.864, Z 13.600} C_DIS
   LIN {X 8.619, Y -3.543, Z 13.600} C_DIS
   LIN {X 8.796, Y -1.533, Z 13.600} C_DIS
   LIN {X 8.838, Y -0.993, Z 13.600} C_DIS
   LIN {X 8.907, Y 0.253, Z 13.600} C_DIS
   LIN {X 9.015, Y 2.109, Z 13.600} C_DIS
   LIN {X 9.033, Y 2.484, Z 13.600} C_DIS
   LIN {X 9.095, Y 4.704, Z 13.600} C_DIS
   LIN {X 9.111, Y 5.424, Z 13.600} C_DIS
   LIN {X 9.099, Y 8.811, Z 13.600} C_DIS
   LIN {X 9.098, Y 9.062, Z 13.600} C_DIS
   LIN {X 9.088, Y 9.441, Z 13.600} C_DIS
   LIN {X 8.974, Y 12.537, Z 13.600} C_DIS
   LIN {X 8.950, Y 12.957, Z 13.600} C_DIS
   LIN {X 8.689, Y 16.541, Z 13.600} C_DIS
   LIN {X 8.581, Y 17.762, Z 13.600} C_DIS
   LIN {X 8.537, Y 18.137, Z 13.600}
   LaserEnd_Ext()
   LIN {X -1.020, Y -30.360, Z 13.600}
   LaserStart_Ext()
   LIN {X -8.010, Y -30.360, Z 13.600}
   LaserEnd_Ext()
   LIN {X -9.569, Y -29.360, Z 13.600}
   LaserStart_Ext()
   LIN {X 0.463, Y -29.360, Z 13.600}
   LaserEnd_Ext()
   LIN {X 1.600, Y -28.360, Z 13.600}
   LaserStart_Ext()
   LIN {X -3.251, Y -28.360, Z 13.600}
   LaserEnd_Ext()
   LIN {X -5.599, Y -28.360, Z 13.600}
   LaserStart_Ext()
   LIN {X -10.594, Y -28.360, Z 13.600}
   LaserEnd_Ext()
   LIN {X -11.301, Y -27.360, Z 13.600}
   LaserStart_Ext()
   LIN {X -7.758, Y -27.360, Z 13.600}
   LaserEnd_Ext()
   LIN {X -1.027, Y -27.360, Z 13.600}
   LaserStart_Ext()
   LIN {X 2.159, Y -27.360, Z 13.600}
   LaserEnd_Ext()
   LIN {X 2.718, Y -26.360, Z 13.600}
   LaserStart_Ext()
   LIN {X -0.286, Y -26.360, Z 13.600}
   LaserEnd_Ext()
   LIN {X -8.759, Y -26.360, Z 13.600}
   LaserStart_Ext()
   LIN {X -11.751, Y -26.360, Z 13.600}
   LaserEnd_Ext()
   LIN {X -12.104, Y -25.360, Z 13.600}
   LaserStart_Ext()
   LIN {X -9.391, Y -25.360, Z 13.600}
   LaserEnd_Ext()
   LIN {X 0.497, Y -25.360, Z 13.600}
   LaserStart_Ext()
   LIN {X 3.257, Y -25.360, Z 13.600}
   LaserEnd_Ext()
   LIN {X 3.556, Y -24.360, Z 13.600}
   LaserStart_Ext()
   LIN {X 0.941, Y -24.360, Z 13.600}
   LaserEnd_Ext()
   LIN {X -9.757, Y -24.360, Z 13.600}
   LaserStart_Ext()
   LIN {X -12.288, Y -24.360, Z 13.600}
   LaserEnd_Ext()
   LIN {X -12.279, Y -23.360, Z 13.600}
   LaserStart_Ext()
   LIN {X -9.874, Y -23.360, Z 13.600}
   LaserEnd_Ext()
   LIN {X 1.116, Y -23.360, Z 13.600}
   LaserStart_Ext()
   LIN {X 3.849, Y -23.360, Z 13.600}
   LaserEnd_Ext()
   LIN {X 4.120, Y -22.360, Z 13.600}
   LaserStart_Ext()
   LIN {X 1.177, Y -22.360, Z 13.600}
   LaserEnd_Ext()
   LIN {X -9.913, Y -22.360, Z 13.600}
   LaserStart_Ext()
   LIN {X -12.274, Y -22.360, Z 13.600}
   LaserEnd_Ext()
   LIN {X -12.169, Y -21.360, Z 13.600}
   LaserStart_Ext()
   LIN {X -9.634, Y -21.360, Z 13.600}
   LaserEnd_Ext()
   LIN {X 0.984, Y -21.360, Z 13.600}
   LaserStart_Ext()
   LIN {X 4.391, Y -21.360, Z 13.600}
   LaserEnd_Ext()
   LIN {X 4.662, Y -20.360, Z 13.600}
   LaserStart_Ext()
   LIN {X 0.583, Y -20.360, Z 13.600}
   LaserEnd_Ext()
   LIN {X -9.249, Y -20.360, Z 13.600}
   LaserStart_Ext()
   LIN {X -11.775, Y -20.360, Z 13.600}
   LaserEnd_Ext()
   LIN {X -11.379, Y -19.360, Z 13.600}
   LaserStart_Ext()
   LIN {X -8.651, Y -19.360, Z 13.600}
   LaserEnd_Ext()
   LIN {X -0.021, Y -19.360, Z 13.600}
   LaserStart_Ext()
   LIN {X 4.914, Y -19.360, Z 13.600}
   LaserEnd_Ext()
   LIN {X 5.158, Y -18.360, Z 13.600}
   LaserStart_Ext()
   LIN {X -1.169, Y -18.360, Z 13.600}
   LaserEnd_Ext()
   LIN {X -7.438, Y -18.360, Z 13.600}
   LaserStart_Ext()
   LIN {X -10.867, Y -18.360, Z 13.600}
   LaserEnd_Ext()
   LIN {X -10.278, Y -17.360, Z 13.600}
   LaserStart_Ext()
   LIN {X -4.453, Y -17.360, Z 13.600}
   LaserEnd_Ext()
   LIN {X -3.620, Y -17.360, Z 13.600}
   LaserStart_Ext()
   LIN {X 5.389, Y -17.360, Z 13.600}
   LaserEnd_Ext()
   LIN {X 5.611, Y -16.360, Z 13.600}
   LaserStart_Ext()
   LIN {X -9.695, Y -16.360, Z 13.600}
   LaserEnd_Ext()
   LIN {X -9.162, Y -15.360, Z 13.600}
   LaserStart_Ext()
   LIN {X 5.810, Y -15.360, Z 13.600}
   LaserEnd_Ext()
   LIN {X 6.009, Y -14.360, Z 13.600}
   LaserStart_Ext()
   LIN {X -8.635, Y -14.360, Z 13.600}
   LaserEnd_Ext()
   LIN {X -8.108, Y -13.360, Z 13.600}
   LaserStart_Ext()
   LIN {X 6.208, Y -13.360, Z 13.600}
   LaserEnd_Ext()
   LIN {X 6.402, Y -12.360, Z 13.600}
   LaserStart_Ext()
   LIN {X -7.636, Y -12.360, Z 13.600}
   LaserEnd_Ext()
   LIN {X -7.169, Y -11.360, Z 13.600}
   LaserStart_Ext()
   LIN {X 6.579, Y -11.360, Z 13.600}
   LaserEnd_Ext()
   LIN {X 6.729, Y -10.360, Z 13.600}
   LaserStart_Ext()
   LIN {X -6.702, Y -10.360, Z 13.600}
   LaserEnd_Ext()
   LIN {X -6.258, Y -9.360, Z 13.600}
   LaserStart_Ext()
   LIN {X 6.880, Y -9.360, Z 13.600}
   LaserEnd_Ext()
   LIN {X 7.035, Y -8.360, Z 13.600}
   LaserStart_Ext()
   LIN {X -5.875, Y -8.360, Z 13.600}
   LaserEnd_Ext()
   LIN {X -5.493, Y -7.360, Z 13.600}
   LaserStart_Ext()
   LIN {X 7.184, Y -7.360, Z 13.600}
   LaserEnd_Ext()
   LIN {X 7.305, Y -6.360, Z 13.600}
   LaserStart_Ext()
   LIN {X -5.110, Y -6.360, Z 13.600}
   LaserEnd_Ext()
   LIN {X -4.727, Y -5.360, Z 13.600}
   LaserStart_Ext()
   LIN {X 7.414, Y -5.360, Z 13.600}
   LaserEnd_Ext()
   LIN {X 7.523, Y -4.360, Z 13.600}
   LaserStart_Ext()
   LIN {X -4.344, Y -4.360, Z 13.600}
   LaserEnd_Ext()
   LIN {X -4.002, Y -3.360, Z 13.600}
   LaserStart_Ext()
   LIN {X 7.631, Y -3.360, Z 13.600}
   LaserEnd_Ext()
   LIN {X 7.719, Y -2.360, Z 13.600}
   LaserStart_Ext()
   LIN {X -3.704, Y -2.360, Z 13.600}
   LaserEnd_Ext()
   LIN {X -3.409, Y -1.360, Z 13.600}
   LaserStart_Ext()
   LIN {X 7.806, Y -1.360, Z 13.600}
   LaserEnd_Ext()
   LIN {X 7.871, Y -0.360, Z 13.600}
   LaserStart_Ext()
   LIN {X -3.116, Y -0.360, Z 13.600}
   LaserEnd_Ext()
   LIN {X -2.824, Y 0.640, Z 13.600}
   LaserStart_Ext()
   LIN {X 7.928, Y 0.640, Z 13.600}
   LaserEnd_Ext()
   LIN {X 7.986, Y 1.640, Z 13.600}
   LaserStart_Ext()
   LIN {X -2.538, Y 1.640, Z 13.600}
   LaserEnd_Ext()
   LIN {X -2.319, Y 2.640, Z 13.600}
   LaserStart_Ext()
   LIN {X 8.037, Y 2.640, Z 13.600}
   LaserEnd_Ext()
   LIN {X 8.065, Y 3.640, Z 13.600}
   LaserStart_Ext()
   LIN {X -2.100, Y 3.640, Z 13.600}
   LaserEnd_Ext()
   LIN {X -1.881, Y 4.640, Z 13.600}
   LaserStart_Ext()
   LIN {X 8.093, Y 4.640, Z 13.600}
   LaserEnd_Ext()
   LIN {X 8.110, Y 5.640, Z 13.600}
   LaserStart_Ext()
   LIN {X -1.660, Y 5.640, Z 13.600}
   LaserEnd_Ext()
   LIN {X -1.465, Y 6.640, Z 13.600}
   LaserStart_Ext()
   LIN {X 8.107, Y 6.640, Z 13.600}
   LaserEnd_Ext()
   LIN {X 8.103, Y 7.640, Z 13.600}
   LaserStart_Ext()
   LIN {X -1.316, Y 7.640, Z 13.600}
   LaserEnd_Ext()
   LIN {X -1.168, Y 8.640, Z 13.600}
   LaserStart_Ext()
   LIN {X 8.100, Y 8.640, Z 13.600}
   LaserEnd_Ext()
   LIN {X 8.080, Y 9.640, Z 13.600}
   LaserStart_Ext()
   LIN {X -1.020, Y 9.640, Z 13.600}
   LaserEnd_Ext()
   LIN {X -0.872, Y 10.640, Z 13.600}
   LaserStart_Ext()
   LIN {X 8.043, Y 10.640, Z 13.600}
   LaserEnd_Ext()
   LIN {X 8.007, Y 11.640, Z 13.600}
   LaserStart_Ext()
   LIN {X -0.736, Y 11.640, Z 13.600}
   LaserEnd_Ext()
   LIN {X -0.648, Y 12.640, Z 13.600}
   LaserStart_Ext()
   LIN {X 7.967, Y 12.640, Z 13.600}
   LaserEnd_Ext()
   LIN {X 7.898, Y 13.640, Z 13.600}
   LaserStart_Ext()
   LIN {X -0.565, Y 13.640, Z 13.600}
   LaserEnd_Ext()
   LIN {X -0.483, Y 14.640, Z 13.600}
   LaserStart_Ext()
   LIN {X 7.825, Y 14.640, Z 13.600}
   LaserEnd_Ext()
   LIN {X 7.752, Y 15.640, Z 13.600}
   LaserStart_Ext()
   LIN {X -0.409, Y 15.640, Z 13.600}
   LaserEnd_Ext()
   LIN {X -0.365, Y 16.640, Z 13.600}
   LaserStart_Ext()
   LIN {X 7.676, Y 16.640, Z 13.600}
   LaserEnd_Ext()
   LIN {X 7.587, Y 17.640, Z 13.600}
   LaserStart_Ext()
   LIN {X -0.337, Y 17.640, Z 13.600}
   LaserEnd_Ext()
   LIN {X -0.336, Y 18.640, Z 13.600}
   LaserStart_Ext()
   LIN {X 7.465, Y 18.640, Z 13.600}
   LaserEnd_Ext()
   LIN {X 7.339, Y 19.640, Z 13.600}
   LaserStart_Ext()
   LIN {X -0.334, Y 19.640, Z 13.600}
   LaserEnd_Ext()
   LIN {X -0.333, Y 20.640, Z 13.600}
   LaserStart_Ext()
   LIN {X 7.212, Y 20.640, Z 13.600}
   LaserEnd_Ext()
   LIN {X 7.093, Y 21.640, Z 13.600}
   LaserStart_Ext()
   LIN {X -0.331, Y 21.640, Z 13.600}
   LaserEnd_Ext()
   LIN {X -0.370, Y 22.640, Z 13.600}
   LaserStart_Ext()
   LIN {X 6.974, Y 22.640, Z 13.600}
   LaserEnd_Ext()
   LIN {X 6.820, Y 23.640, Z 13.600}
   LaserStart_Ext()
   LIN {X -0.427, Y 23.640, Z 13.600}
   LaserEnd_Ext()
   LIN {X -0.484, Y 24.640, Z 13.600}
   LaserStart_Ext()
   LIN {X 6.661, Y 24.640, Z 13.600}
   LaserEnd_Ext()
   LIN {X 6.499, Y 25.640, Z 13.600}
   LaserStart_Ext()
   LIN {X -0.541, Y 25.640, Z 13.600}
   LaserEnd_Ext()
   LIN {X -0.638, Y 26.640, Z 13.600}
   LaserStart_Ext()
   LIN {X 6.304, Y 26.640, Z 13.600}
   LaserEnd_Ext()
   LIN {X 6.110, Y 27.640, Z 13.600}
   LaserStart_Ext()
   LIN {X -0.748, Y 27.640, Z 13.600}
   LaserEnd_Ext()
   LIN {X -0.859, Y 28.640, Z 13.600}
   LaserStart_Ext()
   LIN {X 5.915, Y 28.640, Z 13.600}
   LaserEnd_Ext()
   LIN {X 5.720, Y 29.640, Z 13.600}
   LaserStart_Ext()
   LIN {X -0.974, Y 29.640, Z 13.600}
   LaserEnd_Ext()
   LIN {X -1.127, Y 30.640, Z 13.600}
   LaserStart_Ext()
   LIN {X 5.505, Y 30.640, Z 13.600}
   LaserEnd_Ext()
   LIN {X 5.274, Y 31.640, Z 13.600}
   LaserStart_Ext()
   LIN {X -1.279, Y 31.640, Z 13.600}
   LaserEnd_Ext()
   LIN {X -1.443, Y 32.640, Z 13.600}
   LaserStart_Ext()
   LIN {X 5.043, Y 32.640, Z 13.600}
   LaserEnd_Ext()
   LIN {X 4.794, Y 33.640, Z 13.600}
   LaserStart_Ext()
   LIN {X -1.632, Y 33.640, Z 13.600}
   LaserEnd_Ext()
   LIN {X -1.822, Y 34.640, Z 13.600}
   LaserStart_Ext()
   LIN {X 4.535, Y 34.640, Z 13.600}
   LaserEnd_Ext()
   LIN {X 4.277, Y 35.640, Z 13.600}
   LaserStart_Ext()
   LIN {X -2.039, Y 35.640, Z 13.600}
   LaserEnd_Ext()
   LIN {X -2.262, Y 36.640, Z 13.600}
   LaserStart_Ext()
   LIN {X 3.999, Y 36.640, Z 13.600}
   LaserEnd_Ext()
   LIN {X 3.716, Y 37.640, Z 13.600}
   LaserStart_Ext()
   LIN {X -2.458, Y 37.640, Z 13.600}
   LaserEnd_Ext()
   LIN {X -2.468, Y 38.640, Z 13.600}
   LaserStart_Ext()
   LIN {X 3.418, Y 38.640, Z 13.600}
   LaserEnd_Ext()
   LIN {X 2.966, Y 39.640, Z 13.600}
   LaserStart_Ext()
   LIN {X -2.160, Y 39.640, Z 13.600}
   LaserEnd_Ext()
   LIN {X -1.014, Y 40.640, Z 13.600}
   LaserStart_Ext()
   LIN {X 2.001, Y 40.640, Z 13.600}
   LaserEnd_Ext()
   LIN {X 0.556, Y -22.367, Z 14.450}
   LaserStart_Ext()
   LIN {X 0.576, Y -22.799, Z 14.450} C_DIS
   LIN {X 0.371, Y -24.573, Z 14.450} C_DIS
   LIN {X 0.205, Y -25.047, Z 14.450} C_DIS
   LIN {X -0.968, Y -26.756, Z 14.450} C_DIS
   LIN {X -1.169, Y -26.948, Z 14.450} C_DIS
   LIN {X -2.234, Y -27.641, Z 14.450} C_DIS
   LIN {X -2.444, Y -27.745, Z 14.450} C_DIS
   LIN {X -3.685, Y -28.093, Z 14.450} C_DIS
   LIN {X -3.835, Y -28.116, Z 14.450} C_DIS
   LIN {X -4.810, Y -28.135, Z 14.450} C_DIS
   LIN {X -5.364, Y -28.063, Z 14.450} C_DIS
   LIN {X -5.467, Y -28.043, Z 14.450} C_DIS
   LIN {X -5.701, Y -27.987, Z 14.450} C_DIS
   LIN {X -5.840, Y -27.950, Z 14.450} C_DIS
   LIN {X -6.011, Y -27.896, Z 14.450} C_DIS
   LIN {X -6.205, Y -27.828, Z 14.450} C_DIS
   LIN {X -6.402, Y -27.749, Z 14.450} C_DIS
   LIN {X -6.511, Y -27.700, Z 14.450} C_DIS
   LIN {X -6.604, Y -27.656, Z 14.450} C_DIS
   LIN {X -6.698, Y -27.609, Z 14.450} C_DIS
   LIN {X -6.806, Y -27.552, Z 14.450} C_DIS
   LIN {X -6.894, Y -27.503, Z 14.450} C_DIS
   LIN {X -7.011, Y -27.434, Z 14.450} C_DIS
   LIN {X -7.183, Y -27.323, Z 14.450} C_DIS
   LIN {X -7.343, Y -27.211, Z 14.450} C_DIS
   LIN {X -7.438, Y -27.138, Z 14.450} C_DIS
   LIN {X -7.787, Y -26.846, Z 14.450} C_DIS
   LIN {X -7.889, Y -26.745, Z 14.450} C_DIS
   LIN {X -8.466, Y -26.076, Z 14.450} C_DIS
   LIN {X -8.554, Y -25.941, Z 14.450} C_DIS
   LIN {X -9.183, Y -24.631, Z 14.450} C_DIS
   LIN {X -9.222, Y -24.459, Z 14.450} C_DIS
   LIN {X -9.332, Y -22.528, Z 14.450} C_DIS
   LIN {X -9.267, Y -22.131, Z 14.450} C_DIS
   LIN {X -8.449, Y -20.320, Z 14.450} C_DIS
   LIN {X -8.058, Y -19.803, Z 14.450} C_DIS
   LIN {X -6.640, Y -18.745, Z 14.450} C_DIS
   LIN {X -5.922, Y -18.423, Z 14.450} C_DIS
   LIN {X -4.373, Y -18.189, Z 14.450} C_DIS
   LIN {X -3.310, Y -18.335, Z 14.450} C_DIS
   LIN {X -2.183, Y -18.645, Z 14.450} C_DIS
   LIN {X -1.257, Y -19.324, Z 14.450} C_DIS
   LIN {X -0.504, Y -20.027, Z 14.450} C_DIS
   LIN {X 0.082, Y -20.887, Z 14.450} C_DIS
   LIN {X 0.279, Y -21.400, Z 14.450} C_DIS
   LIN {X 0.556, Y -22.367, Z 14.450}
   LaserEnd_Ext()
   LIN {X 8.282, Y -6.770, Z 14.450}
   LaserStart_Ext()
   LIN {X 8.686, Y -3.067, Z 14.450} C_DIS
   LIN {X 8.739, Y -2.471, Z 14.450} C_DIS
   LIN {X 8.856, Y -0.972, Z 14.450} C_DIS
   LIN {X 9.033, Y 2.236, Z 14.450} C_DIS
   LIN {X 9.110, Y 4.993, Z 14.450} C_DIS
   LIN {X 9.101, Y 8.984, Z 14.450} C_DIS
   LIN {X 9.083, Y 9.451, Z 14.450} C_DIS
   LIN {X 8.969, Y 12.538, Z 14.450} C_DIS
   LIN {X 8.819, Y 14.550, Z 14.450} C_DIS
   LIN {X 8.645, Y 16.931, Z 14.450} C_DIS
   LIN {X 8.609, Y 17.336, Z 14.450} C_DIS
   LIN {X 8.595, Y 17.460, Z 14.450} C_DIS
   LIN {X 8.481, Y 18.360, Z 14.450} C_DIS
   LIN {X 8.023, Y 22.220, Z 14.450} C_DIS
   LIN {X 7.610, Y 24.891, Z 14.450} C_DIS
   LIN {X 7.507, Y 25.533, Z 14.450} C_DIS
   LIN {X 6.914, Y 28.579, Z 14.450} C_DIS
   LIN {X 6.659, Y 29.910, Z 14.450} C_DIS
   LIN {X 6.605, Y 30.161, Z 14.450} C_DIS
   LIN {X 6.306, Y 31.442, Z 14.450} C_DIS
   LIN {X 5.860, Y 33.369, Z 14.450} C_DIS
   LIN {X 5.597, Y 34.386, Z 14.450} C_DIS
   LIN {X 5.145, Y 36.106, Z 14.450} C_DIS
   LIN {X 4.680, Y 37.741, Z 14.450} C_DIS
   LIN {X 4.614, Y 37.972, Z 14.450} C_DIS
   LIN {X 4.529, Y 38.253, Z 14.450} C_DIS
   LIN {X 4.186, Y 39.394, Z 14.450} C_DIS
   LIN {X 3.806, Y 40.123, Z 14.450} C_DIS
   LIN {X 3.503, Y 40.700, Z 14.450} C_DIS
   LIN {X 2.771, Y 41.299, Z 14.450} C_DIS
   LIN {X 2.155, Y 41.806, Z 14.450} C_DIS
   LIN {X 1.612, Y 41.945, Z 14.450} C_DIS
   LIN {X 0.460, Y 42.236, Z 14.450} C_DIS
   LIN {X -0.044, Y 42.146, Z 14.450} C_DIS
   LIN {X -1.690, Y 41.632, Z 14.450} C_DIS
   LIN {X -2.146, Y 41.352, Z 14.450} C_DIS
   LIN {X -2.605, Y 40.805, Z 14.450} C_DIS
   LIN {X -3.162, Y 40.120, Z 14.450} C_DIS
   LIN {X -3.601, Y 38.643, Z 14.450} C_DIS
   LIN {X -3.534, Y 37.818, Z 14.450} C_DIS
   LIN {X -3.492, Y 37.289, Z 14.450} C_DIS
   LIN {X -3.416, Y 36.967, Z 14.450} C_DIS
   LIN {X -3.207, Y 36.070, Z 14.450} C_DIS
   LIN {X -2.901, Y 34.679, Z 14.450} C_DIS
   LIN {X -2.863, Y 34.507, Z 14.450} C_DIS
   LIN {X -2.801, Y 34.178, Z 14.450} C_DIS
   LIN {X -2.417, Y 32.178, Z 14.450} C_DIS
   LIN {X -2.127, Y 30.312, Z 14.450} C_DIS
   LIN {X -1.975, Y 29.316, Z 14.450} C_DIS
   LIN {X -1.952, Y 29.097, Z 14.450} C_DIS
   LIN {X -1.584, Y 25.768, Z 14.450} C_DIS
   LIN {X -1.417, Y 22.854, Z 14.450} C_DIS
   LIN {X -1.357, Y 21.806, Z 14.450} C_DIS
   LIN {X -1.358, Y 17.718, Z 14.450} C_DIS
   LIN {X -1.371, Y 16.957, Z 14.450} C_DIS
   LIN {X -1.407, Y 16.459, Z 14.450} C_DIS
   LIN {X -1.452, Y 15.250, Z 14.450} C_DIS
   LIN {X -1.746, Y 11.709, Z 14.450} C_DIS
   LIN {X -2.496, Y 6.549, Z 14.450} C_DIS
   LIN {X -2.659, Y 5.731, Z 14.450} C_DIS
   LIN {X -3.502, Y 1.883, Z 14.450} C_DIS
   LIN {X -4.855, Y -2.735, Z 14.450} C_DIS
   LIN {X -5.133, Y -3.673, Z 14.450} C_DIS
   LIN {X -7.214, Y -9.099, Z 14.450} C_DIS
   LIN {X -7.340, Y -9.418, Z 14.450} C_DIS
   LIN {X -7.891, Y -10.592, Z 14.450} C_DIS
   LIN {X -9.074, Y -13.124, Z 14.450} C_DIS
   LIN {X -9.572, Y -14.068, Z 14.450} C_DIS
   LIN {X -10.499, Y -15.820, Z 14.450} C_DIS
   LIN {X -11.854, Y -18.143, Z 14.450} C_DIS
   LIN {X -12.057, Y -18.486, Z 14.450} C_DIS
   LIN {X -12.239, Y -18.946, Z 14.450} C_DIS
   LIN {X -13.215, Y -21.437, Z 14.450} C_DIS
   LIN {X -13.185, Y -24.259, Z 14.450} C_DIS
   LIN {X -13.193, Y -25.078, Z 14.450} C_DIS
   LIN {X -13.022, Y -25.579, Z 14.450} C_DIS
   LIN {X -12.247, Y -27.596, Z 14.450} C_DIS
   LIN {X -11.884, Y -28.147, Z 14.450} C_DIS
   LIN {X -11.219, Y -29.037, Z 14.450} C_DIS
   LIN {X -11.107, Y -29.192, Z 14.450} C_DIS
   LIN {X -10.995, Y -29.294, Z 14.450} C_DIS
   LIN {X -10.081, Y -30.155, Z 14.450} C_DIS
   LIN {X -9.522, Y -30.568, Z 14.450} C_DIS
   LIN {X -8.382, Y -31.242, Z 14.450} C_DIS
   LIN {X -8.258, Y -31.309, Z 14.450} C_DIS
   LIN {X -8.114, Y -31.359, Z 14.450} C_DIS
   LIN {X -6.701, Y -31.872, Z 14.450} C_DIS
   LIN {X -6.378, Y -31.937, Z 14.450} C_DIS
   LIN {X -5.055, Y -32.141, Z 14.450} C_DIS
   LIN {X -1.660, Y -31.693, Z 14.450} C_DIS
   LIN {X -1.514, Y -31.679, Z 14.450} C_DIS
   LIN {X 0.346, Y -30.797, Z 14.450} C_DIS
   LIN {X 1.824, Y -29.551, Z 14.450} C_DIS
   LIN {X 2.489, Y -28.946, Z 14.450} C_DIS
   LIN {X 3.318, Y -27.413, Z 14.450} C_DIS
   LIN {X 4.239, Y -25.763, Z 14.450} C_DIS
   LIN {X 4.541, Y -24.755, Z 14.450} C_DIS
   LIN {X 4.873, Y -23.607, Z 14.450} C_DIS
   LIN {X 5.633, Y -20.767, Z 14.450} C_DIS
   LIN {X 5.837, Y -20.014, Z 14.450} C_DIS
   LIN {X 5.909, Y -19.722, Z 14.450} C_DIS
   LIN {X 6.615, Y -16.670, Z 14.450} C_DIS
   LIN {X 7.124, Y -14.112, Z 14.450} C_DIS
   LIN {X 7.593, Y -11.586, Z 14.450} C_DIS
   LIN {X 8.185, Y -7.634, Z 14.450} C_DIS
   LIN {X 8.204, Y -7.495, Z 14.450} C_DIS
   LIN {X 8.282, Y -6.770, Z 14.450}
   LaserEnd_Ext()
   LIN {X 7.602, Y -3.785, Z 14.450}
   LaserStart_Ext()
   LIN {X 7.602, Y 17.341, Z 14.450}
   LaserEnd_Ext()
   LIN {X 6.602, Y 24.859, Z 14.450}
   LaserStart_Ext()
   LIN {X 6.602, Y -11.446, Z 14.450}
   LaserEnd_Ext()
   LIN {X 5.602, Y -16.613, Z 14.450}
   LaserStart_Ext()
   LIN {X 5.602, Y 30.059, Z 14.450}
   LaserEnd_Ext()
   LIN {X 4.602, Y 34.237, Z 14.450}
   LaserStart_Ext()
   LIN {X 4.602, Y -20.751, Z 14.450}
   LaserEnd_Ext()
   LIN {X 3.602, Y -24.404, Z 14.450}
   LaserStart_Ext()
   LIN {X 3.602, Y 37.864, Z 14.450}
   LaserEnd_Ext()
   LIN {X 2.602, Y 40.145, Z 14.450}
   LaserStart_Ext()
   LIN {X 2.602, Y -26.644, Z 14.450}
   LaserEnd_Ext()
   LIN {X 1.602, Y -28.401, Z 14.450}
   LaserStart_Ext()
   LIN {X 1.602, Y 40.915, Z 14.450}
   LaserEnd_Ext()
   LIN {X 0.602, Y 41.169, Z 14.450}
   LaserStart_Ext()
   LIN {X 0.602, Y -19.874, Z 14.450}
   LaserEnd_Ext()
   LIN {X 0.602, Y -26.236, Z 14.450}
   LaserStart_Ext()
   LIN {X 0.602, Y -29.273, Z 14.450}
   LaserEnd_Ext()
   LIN {X -0.398, Y -30.044, Z 14.450}
   LaserStart_Ext()
   LIN {X -0.398, Y -27.595, Z 14.450}
   LaserEnd_Ext()
   LIN {X -0.398, Y -18.758, Z 14.450}
   LaserStart_Ext()
   LIN {X -0.398, Y 16.542, Z 14.450}
   LaserEnd_Ext()
   LIN {X -0.398, Y 22.547, Z 14.450}
   LaserStart_Ext()
   LIN {X -0.398, Y 40.988, Z 14.450}
   LaserEnd_Ext()
   LIN {X -1.398, Y 40.638, Z 14.450}
   LaserStart_Ext()
   LIN {X -1.398, Y 32.134, Z 14.450}
   LaserEnd_Ext()
   LIN {X -1.398, Y 7.152, Z 14.450}
   LaserStart_Ext()
   LIN {X -1.398, Y -17.980, Z 14.450}
   LaserEnd_Ext()
   LIN {X -1.398, Y -28.290, Z 14.450}
   LaserStart_Ext()
   LIN {X -1.398, Y -30.521, Z 14.450}
   LaserEnd_Ext()
   LIN {X -2.398, Y -30.782, Z 14.450}
   LaserStart_Ext()
   LIN {X -2.398, Y -28.770, Z 14.450}
   LaserEnd_Ext()
   LIN {X -2.398, Y -17.548, Z 14.450}
   LaserStart_Ext()
   LIN {X -2.398, Y 2.250, Z 14.450}
   LaserEnd_Ext()
   LIN {X -2.398, Y 37.005, Z 14.450}
   LaserStart_Ext()
   LIN {X -2.398, Y 39.181, Z 14.450}
   LaserEnd_Ext()
   LIN {X -3.398, Y -1.319, Z 14.450}
   LaserStart_Ext()
   LIN {X -3.398, Y -17.314, Z 14.450}
   LaserEnd_Ext()
   LIN {X -3.398, Y -29.051, Z 14.450}
   LaserStart_Ext()
   LIN {X -3.398, Y -30.914, Z 14.450}
   LaserEnd_Ext()
   LIN {X -4.398, Y -31.046, Z 14.450}
   LaserStart_Ext()
   LIN {X -4.398, Y -29.127, Z 14.450}
   LaserEnd_Ext()
   LIN {X -4.398, Y -17.190, Z 14.450}
   LaserStart_Ext()
   LIN {X -4.398, Y -4.549, Z 14.450}
   LaserEnd_Ext()
   LIN {X -5.398, Y -7.158, Z 14.450}
   LaserStart_Ext()
   LIN {X -5.398, Y -17.332, Z 14.450}
   LaserEnd_Ext()
   LIN {X -5.398, Y -29.068, Z 14.450}
   LaserStart_Ext()
   LIN {X -5.398, Y -31.076, Z 14.450}
   LaserEnd_Ext()
   LIN {X -6.398, Y -30.913, Z 14.450}
   LaserStart_Ext()
   LIN {X -6.398, Y -28.821, Z 14.450}
   LaserEnd_Ext()
   LIN {X -6.398, Y -17.540, Z 14.450}
   LaserStart_Ext()
   LIN {X -6.398, Y -9.755, Z 14.450}
   LaserEnd_Ext()
   LIN {X -7.398, Y -11.899, Z 14.450}
   LaserStart_Ext()
   LIN {X -7.398, Y -18.063, Z 14.450}
   LaserEnd_Ext()
   LIN {X -7.398, Y -28.367, Z 14.450}
   LaserStart_Ext()
   LIN {X -7.398, Y -30.555, Z 14.450}
   LaserEnd_Ext()
   LIN {X -8.398, Y -30.071, Z 14.450}
   LaserStart_Ext()
   LIN {X -8.398, Y -27.638, Z 14.450}
   LaserEnd_Ext()
   LIN {X -8.398, Y -18.809, Z 14.450}
   LaserStart_Ext()
   LIN {X -8.398, Y -13.986, Z 14.450}
   LaserEnd_Ext()
   LIN {X -9.398, Y -15.877, Z 14.450}
   LaserStart_Ext()
   LIN {X -9.398, Y -19.992, Z 14.450}
   LaserEnd_Ext()
   LIN {X -9.398, Y -26.476, Z 14.450}
   LaserStart_Ext()
   LIN {X -9.398, Y -29.416, Z 14.450}
   LaserEnd_Ext()
   LIN {X -10.398, Y -28.466, Z 14.450}
   LaserStart_Ext()
   LIN {X -10.398, Y -17.631, Z 14.450}
   LaserEnd_Ext()
   LIN {X -11.398, Y -19.541, Z 14.450}
   LaserStart_Ext()
   LIN {X -11.398, Y -27.018, Z 14.450}
   LaserEnd_Ext()
   LIN {X -1.749, Y -18.866, Z 15.300}
   LaserStart_Ext()
   LIN {X -0.132, Y -20.375, Z 15.300} C_DIS
   LIN {X 0.056, Y -20.652, Z 15.300} C_DIS
   LIN {X 0.504, Y -21.820, Z 15.300} C_DIS
   LIN {X 0.606, Y -22.177, Z 15.300} C_DIS
   LIN {X 0.656, Y -23.241, Z 15.300} C_DIS
   LIN {X 0.572, Y -23.970, Z 15.300} C_DIS
   LIN {X 0.065, Y -25.416, Z 15.300} C_DIS
   LIN {X -0.577, Y -26.351, Z 15.300} C_DIS
   LIN {X -1.444, Y -27.180, Z 15.300} C_DIS
   LIN {X -1.528, Y -27.235, Z 15.300} C_DIS
   LIN {X -2.789, Y -27.859, Z 15.300} C_DIS
   LIN {X -2.976, Y -27.911, Z 15.300} C_DIS
   LIN {X -4.211, Y -28.100, Z 15.300} C_DIS
   LIN {X -4.391, Y -28.104, Z 15.300} C_DIS
   LIN {X -4.549, Y -28.091, Z 15.300} C_DIS
   LIN {X -5.285, Y -28.017, Z 15.300} C_DIS
   LIN {X -5.479, Y -27.980, Z 15.300} C_DIS
   LIN {X -5.766, Y -27.902, Z 15.300} C_DIS
   LIN {X -5.929, Y -27.853, Z 15.300} C_DIS
   LIN {X -6.225, Y -27.746, Z 15.300} C_DIS
   LIN {X -6.452, Y -27.647, Z 15.300} C_DIS
   LIN {X -6.612, Y -27.568, Z 15.300} C_DIS
   LIN {X -6.779, Y -27.481, Z 15.300} C_DIS
   LIN {X -6.911, Y -27.400, Z 15.300} C_DIS
   LIN {X -7.095, Y -27.288, Z 15.300} C_DIS
   LIN {X -7.179, Y -27.230, Z 15.300} C_DIS
   LIN {X -7.354, Y -27.099, Z 15.300} C_DIS
   LIN {X -7.577, Y -26.923, Z 15.300} C_DIS
   LIN {X -8.099, Y -26.397, Z 15.300} C_DIS
   LIN {X -8.198, Y -26.271, Z 15.300} C_DIS
   LIN {X -8.682, Y -25.527, Z 15.300} C_DIS
   LIN {X -9.042, Y -24.777, Z 15.300} C_DIS
   LIN {X -9.221, Y -23.995, Z 15.300} C_DIS
   LIN {X -9.282, Y -22.930, Z 15.300} C_DIS
   LIN {X -9.076, Y -21.675, Z 15.300} C_DIS
   LIN {X -8.659, Y -20.750, Z 15.300} C_DIS
   LIN {X -7.680, Y -19.459, Z 15.300} C_DIS
   LIN {X -7.029, Y -18.973, Z 15.300} C_DIS
   LIN {X -5.444, Y -18.262, Z 15.300} C_DIS
   LIN {X -4.797, Y -18.164, Z 15.300} C_DIS
   LIN {X -2.571, Y -18.470, Z 15.300} C_DIS
   LIN {X -2.120, Y -18.594, Z 15.300} C_DIS
   LIN {X -1.749, Y -18.866, Z 15.300}
   LaserEnd_Ext()
   LIN {X -2.263, Y 41.366, Z 15.300}
   LaserStart_Ext()
   LIN {X -1.857, Y 41.617, Z 15.300} C_DIS
   LIN {X -1.463, Y 41.860, Z 15.300} C_DIS
   LIN {X -0.692, Y 42.100, Z 15.300} C_DIS
   LIN {X 0.369, Y 42.290, Z 15.300} C_DIS
   LIN {X 2.079, Y 41.866, Z 15.300} C_DIS
   LIN {X 2.727, Y 41.340, Z 15.300} C_DIS
   LIN {X 3.430, Y 40.764, Z 15.300} C_DIS
   LIN {X 3.859, Y 39.946, Z 15.300} C_DIS
   LIN {X 4.116, Y 39.460, Z 15.300} C_DIS
   LIN {X 4.249, Y 39.023, Z 15.300} C_DIS
   LIN {X 4.547, Y 38.038, Z 15.300} C_DIS
   LIN {X 5.048, Y 36.297, Z 15.300} C_DIS
   LIN {X 5.077, Y 36.193, Z 15.300} C_DIS
   LIN {X 5.160, Y 35.878, Z 15.300} C_DIS
   LIN {X 5.795, Y 33.475, Z 15.300} C_DIS
   LIN {X 6.081, Y 32.269, Z 15.300} C_DIS
   LIN {X 6.544, Y 30.286, Z 15.300} C_DIS
   LIN {X 6.765, Y 29.249, Z 15.300} C_DIS
   LIN {X 7.403, Y 25.928, Z 15.300} C_DIS
   LIN {X 7.491, Y 25.468, Z 15.300} C_DIS
   LIN {X 7.586, Y 24.859, Z 15.300} C_DIS
   LIN {X 8.082, Y 21.649, Z 15.300} C_DIS
   LIN {X 8.576, Y 17.491, Z 15.300} C_DIS
   LIN {X 8.622, Y 17.079, Z 15.300} C_DIS
   LIN {X 8.680, Y 16.331, Z 15.300} C_DIS
   LIN {X 8.968, Y 12.484, Z 15.300} C_DIS
   LIN {X 9.050, Y 10.271, Z 15.300} C_DIS
   LIN {X 9.108, Y 8.768, Z 15.300} C_DIS
   LIN {X 9.117, Y 5.447, Z 15.300} C_DIS
   LIN {X 9.073, Y 3.717, Z 15.300} C_DIS
   LIN {X 9.013, Y 1.560, Z 15.300} C_DIS
   LIN {X 8.875, Y -0.950, Z 15.300} C_DIS
   LIN {X 8.746, Y -2.590, Z 15.300} C_DIS
   LIN {X 8.687, Y -3.289, Z 15.300} C_DIS
   LIN {X 8.286, Y -7.020, Z 15.300} C_DIS
   LIN {X 8.039, Y -8.851, Z 15.300} C_DIS
   LIN {X 7.657, Y -11.404, Z 15.300} C_DIS
   LIN {X 6.929, Y -15.323, Z 15.300} C_DIS
   LIN {X 6.696, Y -16.491, Z 15.300} C_DIS
   LIN {X 6.301, Y -18.201, Z 15.300} C_DIS
   LIN {X 5.941, Y -19.786, Z 15.300} C_DIS
   LIN {X 5.722, Y -20.651, Z 15.300} C_DIS
   LIN {X 5.040, Y -23.202, Z 15.300} C_DIS
   LIN {X 4.332, Y -25.653, Z 15.300} C_DIS
   LIN {X 2.642, Y -28.801, Z 15.300} C_DIS
   LIN {X 1.275, Y -30.045, Z 15.300} C_DIS
   LIN {X 0.482, Y -30.713, Z 15.300} C_DIS
   LIN {X -0.548, Y -31.204, Z 15.300} C_DIS
   LIN {X -1.656, Y -31.689, Z 15.300} C_DIS
   LIN {X -3.163, Y -31.877, Z 15.300} C_DIS
   LIN {X -4.877, Y -32.103, Z 15.300} C_DIS
   LIN {X -5.792, Y -31.962, Z 15.300} C_DIS
   LIN {X -6.681, Y -31.814, Z 15.300} C_DIS
   LIN {X -7.317, Y -31.590, Z 15.300} C_DIS
   LIN {X -8.644, Y -31.025, Z 15.300} C_DIS
   LIN {X -9.579, Y -30.435, Z 15.300} C_DIS
   LIN {X -9.848, Y -30.244, Z 15.300} C_DIS
   LIN {X -9.941, Y -30.158, Z 15.300} C_DIS
   LIN {X -10.951, Y -29.237, Z 15.300} C_DIS
   LIN {X -11.953, Y -27.861, Z 15.300} C_DIS
   LIN {X -12.137, Y -27.618, Z 15.300} C_DIS
   LIN {X -12.196, Y -27.478, Z 15.300} C_DIS
   LIN {X -13.104, Y -25.123, Z 15.300} C_DIS
   LIN {X -13.118, Y -24.157, Z 15.300} C_DIS
   LIN {X -13.146, Y -21.412, Z 15.300} C_DIS
   LIN {X -12.382, Y -19.461, Z 15.300} C_DIS
   LIN {X -11.995, Y -18.458, Z 15.300} C_DIS
   LIN {X -11.411, Y -17.449, Z 15.300} C_DIS
   LIN {X -10.467, Y -15.830, Z 15.300} C_DIS
   LIN {X -9.307, Y -13.640, Z 15.300} C_DIS
   LIN {X -9.185, Y -13.410, Z 15.300} C_DIS
   LIN {X -7.374, Y -9.556, Z 15.300} C_DIS
   LIN {X -6.918, Y -8.408, Z 15.300} C_DIS
   LIN {X -5.263, Y -4.090, Z 15.300} C_DIS
   LIN {X -4.456, Y -1.371, Z 15.300} C_DIS
   LIN {X -3.475, Y 1.978, Z 15.300} C_DIS
   LIN {X -2.864, Y 4.768, Z 15.300} C_DIS
   LIN {X -2.458, Y 6.809, Z 15.300} C_DIS
   LIN {X -1.834, Y 11.090, Z 15.300} C_DIS
   LIN {X -1.756, Y 11.728, Z 15.300} C_DIS
   LIN {X -1.513, Y 14.657, Z 15.300} C_DIS
   LIN {X -1.475, Y 15.657, Z 15.300} C_DIS
   LIN {X -1.403, Y 16.648, Z 15.300} C_DIS
   LIN {X -1.379, Y 18.163, Z 15.300} C_DIS
   LIN {X -1.378, Y 21.592, Z 15.300} C_DIS
   LIN {X -1.543, Y 24.460, Z 15.300} C_DIS
   LIN {X -1.614, Y 25.711, Z 15.300} C_DIS
   LIN {X -1.838, Y 27.737, Z 15.300} C_DIS
   LIN {X -2.021, Y 29.367, Z 15.300} C_DIS
   LIN {X -2.376, Y 31.622, Z 15.300} C_DIS
   LIN {X -2.470, Y 32.227, Z 15.300} C_DIS
   LIN {X -2.538, Y 32.581, Z 15.300} C_DIS
   LIN {X -2.921, Y 34.556, Z 15.300} C_DIS
   LIN {X -3.237, Y 35.979, Z 15.300} C_DIS
   LIN {X -3.269, Y 36.118, Z 15.300} C_DIS
   LIN {X -3.311, Y 36.294, Z 15.300} C_DIS
   LIN {X -3.557, Y 37.336, Z 15.300} C_DIS
   LIN {X -3.618, Y 38.113, Z 15.300} C_DIS
   LIN {X -3.664, Y 38.741, Z 15.300} C_DIS
   LIN {X -3.454, Y 39.447, Z 15.300} C_DIS
   LIN {X -3.248, Y 40.139, Z 15.300} C_DIS
   LIN {X -2.781, Y 40.713, Z 15.300} C_DIS
   LIN {X -2.263, Y 41.366, Z 15.300}
   LaserEnd_Ext()
   LIN {X 2.147, Y 40.522, Z 15.300}
   LaserStart_Ext()
   LIN {X -1.656, Y 40.522, Z 15.300}
   LaserEnd_Ext()
   LIN {X -2.388, Y 39.522, Z 15.300}
   LaserStart_Ext()
   LIN {X 2.952, Y 39.522, Z 15.300}
   LaserEnd_Ext()
   LIN {X 3.356, Y 38.522, Z 15.300}
   LaserStart_Ext()
   LIN {X -2.645, Y 38.522, Z 15.300}
   LaserEnd_Ext()
   LIN {X -2.568, Y 37.522, Z 15.300}
   LaserStart_Ext()
   LIN {X 3.655, Y 37.522, Z 15.300}
   LaserEnd_Ext()
   LIN {X 3.943, Y 36.522, Z 15.300}
   LaserStart_Ext()
   LIN {X -2.337, Y 36.522, Z 15.300}
   LaserEnd_Ext()
   LIN {X -2.112, Y 35.522, Z 15.300}
   LaserStart_Ext()
   LIN {X 4.220, Y 35.522, Z 15.300}
   LaserEnd_Ext()
   LIN {X 4.484, Y 34.522, Z 15.300}
   LaserStart_Ext()
   LIN {X -1.896, Y 34.522, Z 15.300}
   LaserEnd_Ext()
   LIN {X -1.702, Y 33.522, Z 15.300}
   LaserStart_Ext()
   LIN {X 4.748, Y 33.522, Z 15.300}
   LaserEnd_Ext()
   LIN {X 4.993, Y 32.522, Z 15.300}
   LaserStart_Ext()
   LIN {X -1.508, Y 32.522, Z 15.300}
   LaserEnd_Ext()
   LIN {X -1.348, Y 31.522, Z 15.300}
   LaserStart_Ext()
   LIN {X 5.229, Y 31.522, Z 15.300}
   LaserEnd_Ext()
   LIN {X 5.462, Y 30.522, Z 15.300}
   LaserStart_Ext()
   LIN {X -1.190, Y 30.522, Z 15.300}
   LaserEnd_Ext()
   LIN {X -1.033, Y 29.522, Z 15.300}
   LaserStart_Ext()
   LIN {X 5.685, Y 29.522, Z 15.300}
   LaserEnd_Ext()
   LIN {X 5.887, Y 28.522, Z 15.300}
   LaserStart_Ext()
   LIN {X -0.920, Y 28.522, Z 15.300}
   LaserEnd_Ext()
   LIN {X -0.808, Y 27.522, Z 15.300}
   LaserStart_Ext()
   LIN {X 6.079, Y 27.522, Z 15.300}
   LaserEnd_Ext()
   LIN {X 6.271, Y 26.522, Z 15.300}
   LaserStart_Ext()
   LIN {X -0.698, Y 26.522, Z 15.300}
   LaserEnd_Ext()
   LIN {X -0.602, Y 25.522, Z 15.300}
   LaserStart_Ext()
   LIN {X 6.463, Y 25.522, Z 15.300}
   LaserEnd_Ext()
   LIN {X 6.626, Y 24.522, Z 15.300}
   LaserStart_Ext()
   LIN {X -0.545, Y 24.522, Z 15.300}
   LaserEnd_Ext()
   LIN {X -0.487, Y 23.522, Z 15.300}
   LaserStart_Ext()
   LIN {X 6.781, Y 23.522, Z 15.300}
   LaserEnd_Ext()
   LIN {X 6.935, Y 22.522, Z 15.300}
   LaserStart_Ext()
   LIN {X -0.430, Y 22.522, Z 15.300}
   LaserEnd_Ext()
   LIN {X -0.378, Y 21.522, Z 15.300}
   LaserStart_Ext()
   LIN {X 7.090, Y 21.522, Z 15.300}
   LaserEnd_Ext()
   LIN {X 7.209, Y 20.522, Z 15.300}
   LaserStart_Ext()
   LIN {X -0.378, Y 20.522, Z 15.300}
   LaserEnd_Ext()
   LIN {X -0.379, Y 19.522, Z 15.300}
   LaserStart_Ext()
   LIN {X 7.328, Y 19.522, Z 15.300}
   LaserEnd_Ext()
   LIN {X 7.447, Y 18.522, Z 15.300}
   LaserStart_Ext()
   LIN {X -0.379, Y 18.522, Z 15.300}
   LaserEnd_Ext()
   LIN {X -0.389, Y 17.522, Z 15.300}
   LaserStart_Ext()
   LIN {X 7.565, Y 17.522, Z 15.300}
   LaserEnd_Ext()
   LIN {X 7.663, Y 16.522, Z 15.300}
   LaserStart_Ext()
   LIN {X -0.410, Y 16.522, Z 15.300}
   LaserEnd_Ext()
   LIN {X -0.480, Y 15.522, Z 15.300}
   LaserStart_Ext()
   LIN {X 7.738, Y 15.522, Z 15.300}
   LaserEnd_Ext()
   LIN {X 7.813, Y 14.522, Z 15.300}
   LaserStart_Ext()
   LIN {X -0.521, Y 14.522, Z 15.300}
   LaserEnd_Ext()
   LIN {X -0.604, Y 13.522, Z 15.300}
   LaserStart_Ext()
   LIN {X 7.888, Y 13.522, Z 15.300}
   LaserEnd_Ext()
   LIN {X 7.962, Y 12.522, Z 15.300}
   LaserStart_Ext()
   LIN {X -0.686, Y 12.522, Z 15.300}
   LaserEnd_Ext()
   LIN {X -0.774, Y 11.522, Z 15.300}
   LaserStart_Ext()
   LIN {X 8.003, Y 11.522, Z 15.300}
   LaserEnd_Ext()
   LIN {X 8.040, Y 10.522, Z 15.300}
   LaserStart_Ext()
   LIN {X -0.906, Y 10.522, Z 15.300}
   LaserEnd_Ext()
   LIN {X -1.052, Y 9.522, Z 15.300}
   LaserStart_Ext()
   LIN {X 8.078, Y 9.522, Z 15.300}
   LaserEnd_Ext()
   LIN {X 8.109, Y 8.522, Z 15.300}
   LaserStart_Ext()
   LIN {X -1.198, Y 8.522, Z 15.300}
   LaserEnd_Ext()
   LIN {X -1.343, Y 7.522, Z 15.300}
   LaserStart_Ext()
   LIN {X 8.111, Y 7.522, Z 15.300}
   LaserEnd_Ext()
   LIN {X 8.114, Y 6.522, Z 15.300}
   LaserStart_Ext()
   LIN {X -1.495, Y 6.522, Z 15.300}
   LaserEnd_Ext()
   LIN {X -1.694, Y 5.522, Z 15.300}
   LaserStart_Ext()
   LIN {X 8.117, Y 5.522, Z 15.300}
   LaserEnd_Ext()
   LIN {X 8.093, Y 4.522, Z 15.300}
   LaserStart_Ext()
   LIN {X -1.894, Y 4.522, Z 15.300}
   LaserEnd_Ext()
   LIN {X -2.113, Y 3.522, Z 15.300}
   LaserStart_Ext()
   LIN {X 8.067, Y 3.522, Z 15.300}
   LaserEnd_Ext()
   LIN {X 8.039, Y 2.522, Z 15.300}
   LaserStart_Ext()
   LIN {X -2.332, Y 2.522, Z 15.300}
   LaserEnd_Ext()
   LIN {X -2.567, Y 1.522, Z 15.300}
   LaserStart_Ext()
   LIN {X 8.009, Y 1.522, Z 15.300}
   LaserEnd_Ext()
   LIN {X 7.954, Y 0.522, Z 15.300}
   LaserStart_Ext()
   LIN {X -2.860, Y 0.522, Z 15.300}
   LaserEnd_Ext()
   LIN {X -3.153, Y -0.478, Z 15.300}
   LaserStart_Ext()
   LIN {X 7.899, Y -0.478, Z 15.300}
   LaserEnd_Ext()
   LIN {X 7.830, Y -1.478, Z 15.300}
   LaserStart_Ext()
   LIN {X -3.445, Y -1.478, Z 15.300}
   LaserEnd_Ext()
   LIN {X -3.741, Y -2.478, Z 15.300}
   LaserStart_Ext()
   LIN {X 7.752, Y -2.478, Z 15.300}
   LaserEnd_Ext()
   LIN {X 7.661, Y -3.478, Z 15.300}
   LaserStart_Ext()
   LIN {X -4.038, Y -3.478, Z 15.300}
   LaserEnd_Ext()
   LIN {X -4.341, Y -4.478, Z 15.300}
   LaserStart_Ext()
   LIN {X 7.553, Y -4.478, Z 15.300}
   LaserEnd_Ext()
   LIN {X 7.446, Y -5.478, Z 15.300}
   LaserStart_Ext()
   LIN {X -4.724, Y -5.478, Z 15.300}
   LaserEnd_Ext()
   LIN {X -5.108, Y -6.478, Z 15.300}
   LaserStart_Ext()
   LIN {X 7.338, Y -6.478, Z 15.300}
   LaserEnd_Ext()
   LIN {X 7.215, Y -7.478, Z 15.300}
   LaserStart_Ext()
   LIN {X -5.491, Y -7.478, Z 15.300}
   LaserEnd_Ext()
   LIN {X -5.874, Y -8.478, Z 15.300}
   LaserStart_Ext()
   LIN {X 7.080, Y -8.478, Z 15.300}
   LaserEnd_Ext()
   LIN {X 6.934, Y -9.478, Z 15.300}
   LaserStart_Ext()
   LIN {X -6.267, Y -9.478, Z 15.300}
   LaserEnd_Ext()
   LIN {X -6.702, Y -10.478, Z 15.300}
   LaserStart_Ext()
   LIN {X 6.784, Y -10.478, Z 15.300}
   LaserEnd_Ext()
   LIN {X 6.626, Y -11.478, Z 15.300}
   LaserStart_Ext()
   LIN {X -7.172, Y -11.478, Z 15.300}
   LaserEnd_Ext()
   LIN {X -7.642, Y -12.478, Z 15.300}
   LaserStart_Ext()
   LIN {X 6.440, Y -12.478, Z 15.300}
   LaserEnd_Ext()
   LIN {X 6.254, Y -13.478, Z 15.300}
   LaserStart_Ext()
   LIN {X -8.111, Y -13.478, Z 15.300}
   LaserEnd_Ext()
   LIN {X -8.620, Y -14.478, Z 15.300}
   LaserStart_Ext()
   LIN {X 6.069, Y -14.478, Z 15.300}
   LaserEnd_Ext()
   LIN {X 5.878, Y -15.478, Z 15.300}
   LaserStart_Ext()
   LIN {X -9.149, Y -15.478, Z 15.300}
   LaserEnd_Ext()
   LIN {X -9.687, Y -16.478, Z 15.300}
   LaserStart_Ext()
   LIN {X 5.673, Y -16.478, Z 15.300}
   LaserEnd_Ext()
   LIN {X 5.442, Y -17.478, Z 15.300}
   LaserStart_Ext()
   LIN {X -2.445, Y -17.478, Z 15.300}
   LaserEnd_Ext()
   LIN {X -6.140, Y -17.478, Z 15.300}
   LaserStart_Ext()
   LIN {X -10.271, Y -17.478, Z 15.300}
   LaserEnd_Ext()
   LIN {X -10.852, Y -18.478, Z 15.300}
   LaserStart_Ext()
   LIN {X -8.038, Y -18.478, Z 15.300}
   LaserEnd_Ext()
   LIN {X -0.699, Y -18.478, Z 15.300}
   LaserStart_Ext()
   LIN {X 5.213, Y -18.478, Z 15.300}
   LaserEnd_Ext()
   LIN {X 4.986, Y -19.478, Z 15.300}
   LaserStart_Ext()
   LIN {X 0.372, Y -19.478, Z 15.300}
   LaserEnd_Ext()
   LIN {X -8.950, Y -19.478, Z 15.300}
   LaserStart_Ext()
   LIN {X -11.317, Y -19.478, Z 15.300}
   LaserEnd_Ext()
   LIN {X -11.707, Y -20.478, Z 15.300}
   LaserStart_Ext()
   LIN {X -9.633, Y -20.478, Z 15.300}
   LaserEnd_Ext()
   LIN {X 1.061, Y -20.478, Z 15.300}
   LaserStart_Ext()
   LIN {X 4.733, Y -20.478, Z 15.300}
   LaserEnd_Ext()
   LIN {X 4.466, Y -21.478, Z 15.300}
   LaserStart_Ext()
   LIN {X 1.443, Y -21.478, Z 15.300}
   LaserEnd_Ext()
   LIN {X -10.056, Y -21.478, Z 15.300}
   LaserStart_Ext()
   LIN {X -12.099, Y -21.478, Z 15.300}
   LaserEnd_Ext()
   LIN {X -12.135, Y -22.478, Z 15.300}
   LaserStart_Ext()
   LIN {X -10.221, Y -22.478, Z 15.300}
   LaserEnd_Ext()
   LIN {X 1.621, Y -22.478, Z 15.300}
   LaserStart_Ext()
   LIN {X 4.199, Y -22.478, Z 15.300}
   LaserEnd_Ext()
   LIN {X 3.919, Y -23.478, Z 15.300}
   LaserStart_Ext()
   LIN {X 1.636, Y -23.478, Z 15.300}
   LaserEnd_Ext()
   LIN {X -10.252, Y -23.478, Z 15.300}
   LaserStart_Ext()
   LIN {X -12.125, Y -23.478, Z 15.300}
   LaserEnd_Ext()
   LIN {X -12.113, Y -24.478, Z 15.300}
   LaserStart_Ext()
   LIN {X -10.136, Y -24.478, Z 15.300}
   LaserEnd_Ext()
   LIN {X 1.454, Y -24.478, Z 15.300}
   LaserStart_Ext()
   LIN {X 3.630, Y -24.478, Z 15.300}
   LaserEnd_Ext()
   LIN {X 3.302, Y -25.478, Z 15.300}
   LaserStart_Ext()
   LIN {X 1.103, Y -25.478, Z 15.300}
   LaserEnd_Ext()
   LIN {X -9.814, Y -25.478, Z 15.300}
   LaserStart_Ext()
   LIN {X -11.895, Y -25.478, Z 15.300}
   LaserEnd_Ext()
   LIN {X -11.509, Y -26.478, Z 15.300}
   LaserStart_Ext()
   LIN {X -9.256, Y -26.478, Z 15.300}
   LaserEnd_Ext()
   LIN {X 0.549, Y -26.478, Z 15.300}
   LaserStart_Ext()
   LIN {X 2.761, Y -26.478, Z 15.300}
   LaserEnd_Ext()
   LIN {X 2.220, Y -27.478, Z 15.300}
   LaserStart_Ext()
   LIN {X -0.309, Y -27.478, Z 15.300}
   LaserEnd_Ext()
   LIN {X -8.435, Y -27.478, Z 15.300}
   LaserStart_Ext()
   LIN {X -10.995, Y -27.478, Z 15.300}
   LaserEnd_Ext()
   LIN {X -10.266, Y -28.478, Z 15.300}
   LaserStart_Ext()
   LIN {X -7.030, Y -28.478, Z 15.300}
   LaserEnd_Ext()
   LIN {X -1.787, Y -28.478, Z 15.300}
   LaserStart_Ext()
   LIN {X 1.511, Y -28.478, Z 15.300}
   LaserEnd_Ext()
   LIN {X 0.395, Y -29.478, Z 15.300}
   LaserStart_Ext()
   LIN {X -9.199, Y -29.478, Z 15.300}
   LaserEnd_Ext()
   LIN {X -7.375, Y -30.478, Z 15.300}
   LaserStart_Ext()
   LIN {X -1.384, Y -30.478, Z 15.300}
   LaserEnd_Ext()
   LIN {X 0.715, Y -23.634, Z 16.150}
   LaserStart_Ext()
   LIN {X 0.229, Y -24.920, Z 16.150} C_DIS
   LIN {X -0.075, Y -25.785, Z 16.150} C_DIS
   LIN {X -0.185, Y -25.946, Z 16.150} C_DIS
   LIN {X -0.357, Y -26.110, Z 16.150} C_DIS
   LIN {X -1.750, Y -27.363, Z 16.150} C_DIS
   LIN {X -2.491, Y -27.725, Z 16.150} C_DIS
   LIN {X -3.087, Y -27.901, Z 16.150} C_DIS
   LIN {X -4.100, Y -28.055, Z 16.150} C_DIS
   LIN {X -4.466, Y -28.052, Z 16.150} C_DIS
   LIN {X -5.178, Y -27.979, Z 16.150} C_DIS
   LIN {X -5.363, Y -27.933, Z 16.150} C_DIS
   LIN {X -5.954, Y -27.775, Z 16.150} C_DIS
   LIN {X -6.060, Y -27.733, Z 16.150} C_DIS
   LIN {X -6.439, Y -27.574, Z 16.150} C_DIS
   LIN {X -6.962, Y -27.273, Z 16.150} C_DIS
   LIN {X -7.059, Y -27.217, Z 16.150} C_DIS
   LIN {X -7.152, Y -27.146, Z 16.150} C_DIS
   LIN {X -7.617, Y -26.774, Z 16.150} C_DIS
   LIN {X -7.877, Y -26.516, Z 16.150} C_DIS
   LIN {X -8.106, Y -26.265, Z 16.150} C_DIS
   LIN {X -8.688, Y -25.301, Z 16.150} C_DIS
   LIN {X -8.810, Y -25.112, Z 16.150} C_DIS
   LIN {X -8.902, Y -24.922, Z 16.150} C_DIS
   LIN {X -9.220, Y -23.532, Z 16.150} C_DIS
   LIN {X -9.231, Y -23.332, Z 16.150} C_DIS
   LIN {X -8.886, Y -21.219, Z 16.150} C_DIS
   LIN {X -8.541, Y -20.748, Z 16.150} C_DIS
   LIN {X -7.402, Y -19.215, Z 16.150} C_DIS
   LIN {X -7.292, Y -19.125, Z 16.150} C_DIS
   LIN {X -5.177, Y -18.163, Z 16.150} C_DIS
   LIN {X -4.912, Y -18.121, Z 16.150} C_DIS
   LIN {X -2.480, Y -18.447, Z 16.150} C_DIS
   LIN {X -2.056, Y -18.544, Z 16.150} C_DIS
   LIN {X -1.663, Y -18.851, Z 16.150} C_DIS
   LIN {X -0.072, Y -20.297, Z 16.150} C_DIS
   LIN {X 0.193, Y -20.744, Z 16.150} C_DIS
   LIN {X 0.607, Y -21.840, Z 16.150} C_DIS
   LIN {X 0.683, Y -22.192, Z 16.150} C_DIS
   LIN {X 0.738, Y -23.446, Z 16.150} C_DIS
   LIN {X 0.715, Y -23.634, Z 16.150}
   LaserEnd_Ext()
   LIN {X 8.800, Y -2.112, Z 16.150}
   LaserStart_Ext()
   LIN {X 8.639, Y -4.021, Z 16.150} C_DIS
   LIN {X 8.368, Y -6.545, Z 16.150} C_DIS
   LIN {X 7.894, Y -10.067, Z 16.150} C_DIS
   LIN {X 7.721, Y -11.222, Z 16.150} C_DIS
   LIN {X 6.928, Y -15.489, Z 16.150} C_DIS
   LIN {X 6.778, Y -16.307, Z 16.150} C_DIS
   LIN {X 6.740, Y -16.487, Z 16.150} C_DIS
   LIN {X 6.031, Y -19.609, Z 16.150} C_DIS
   LIN {X 5.531, Y -21.584, Z 16.150} C_DIS
   LIN {X 5.207, Y -22.797, Z 16.150} C_DIS
   LIN {X 4.870, Y -23.962, Z 16.150} C_DIS
   LIN {X 4.397, Y -25.631, Z 16.150} C_DIS
   LIN {X 3.834, Y -26.734, Z 16.150} C_DIS
   LIN {X 2.794, Y -28.656, Z 16.150} C_DIS
   LIN {X 0.726, Y -30.538, Z 16.150} C_DIS
   LIN {X 0.618, Y -30.629, Z 16.150} C_DIS
   LIN {X 0.478, Y -30.696, Z 16.150} C_DIS
   LIN {X -1.844, Y -31.711, Z 16.150} C_DIS
   LIN {X -4.622, Y -32.058, Z 16.150} C_DIS
   LIN {X -4.746, Y -32.061, Z 16.150} C_DIS
   LIN {X -4.950, Y -32.009, Z 16.150} C_DIS
   LIN {X -6.961, Y -31.655, Z 16.150} C_DIS
   LIN {X -8.722, Y -30.897, Z 16.150} C_DIS
   LIN {X -9.191, Y -30.577, Z 16.150} C_DIS
   LIN {X -10.066, Y -29.955, Z 16.150} C_DIS
   LIN {X -10.584, Y -29.474, Z 16.150} C_DIS
   LIN {X -10.795, Y -29.282, Z 16.150} C_DIS
   LIN {X -11.004, Y -28.995, Z 16.150} C_DIS
   LIN {X -12.009, Y -27.666, Z 16.150} C_DIS
   LIN {X -12.333, Y -26.899, Z 16.150} C_DIS
   LIN {X -13.027, Y -25.097, Z 16.150} C_DIS
   LIN {X -13.071, Y -22.096, Z 16.150} C_DIS
   LIN {X -13.078, Y -21.386, Z 16.150} C_DIS
   LIN {X -12.881, Y -20.882, Z 16.150} C_DIS
   LIN {X -11.934, Y -18.429, Z 16.150} C_DIS
   LIN {X -10.507, Y -15.964, Z 16.150} C_DIS
   LIN {X -10.434, Y -15.840, Z 16.150} C_DIS
   LIN {X -10.346, Y -15.673, Z 16.150} C_DIS
   LIN {X -9.297, Y -13.694, Z 16.150} C_DIS
   LIN {X -8.938, Y -12.952, Z 16.150} C_DIS
   LIN {X -7.408, Y -9.695, Z 16.150} C_DIS
   LIN {X -6.623, Y -7.716, Z 16.150} C_DIS
   LIN {X -5.393, Y -4.507, Z 16.150} C_DIS
   LIN {X -4.057, Y -0.007, Z 16.150} C_DIS
   LIN {X -3.448, Y 2.072, Z 16.150} C_DIS
   LIN {X -3.069, Y 3.805, Z 16.150} C_DIS
   LIN {X -2.419, Y 7.069, Z 16.150} C_DIS
   LIN {X -1.919, Y 10.500, Z 16.150} C_DIS
   LIN {X -1.766, Y 11.746, Z 16.150} C_DIS
   LIN {X -1.574, Y 14.064, Z 16.150} C_DIS
   LIN {X -1.544, Y 14.855, Z 16.150} C_DIS
   LIN {X -1.436, Y 16.339, Z 16.150} C_DIS
   LIN {X -1.400, Y 18.607, Z 16.150} C_DIS
   LIN {X -1.399, Y 21.377, Z 16.150} C_DIS
   LIN {X -1.629, Y 25.379, Z 16.150} C_DIS
   LIN {X -1.650, Y 25.711, Z 16.150} C_DIS
   LIN {X -1.788, Y 26.925, Z 16.150} C_DIS
   LIN {X -2.068, Y 29.417, Z 16.150} C_DIS
   LIN {X -2.234, Y 30.477, Z 16.150} C_DIS
   LIN {X -2.523, Y 32.277, Z 16.150} C_DIS
   LIN {X -2.945, Y 34.426, Z 16.150} C_DIS
   LIN {X -2.980, Y 34.604, Z 16.150} C_DIS
   LIN {X -3.331, Y 36.165, Z 16.150} C_DIS
   LIN {X -3.530, Y 37.003, Z 16.150} C_DIS
   LIN {X -3.621, Y 37.383, Z 16.150} C_DIS
   LIN {X -3.668, Y 38.059, Z 16.150} C_DIS
   LIN {X -3.726, Y 38.838, Z 16.150} C_DIS
   LIN {X -3.544, Y 39.451, Z 16.150} C_DIS
   LIN {X -3.313, Y 40.198, Z 16.150} C_DIS
   LIN {X -2.719, Y 40.952, Z 16.150} C_DIS
   LIN {X -2.380, Y 41.379, Z 16.150} C_DIS
   LIN {X -1.594, Y 41.864, Z 16.150} C_DIS
   LIN {X -1.325, Y 42.032, Z 16.150} C_DIS
   LIN {X -1.112, Y 42.095, Z 16.150} C_DIS
   LIN {X 0.306, Y 42.348, Z 16.150} C_DIS
   LIN {X 1.625, Y 42.021, Z 16.150} C_DIS
   LIN {X 2.003, Y 41.926, Z 16.150} C_DIS
   LIN {X 2.601, Y 41.440, Z 16.150} C_DIS
   LIN {X 3.356, Y 40.828, Z 16.150} C_DIS
   LIN {X 3.582, Y 40.403, Z 16.150} C_DIS
   LIN {X 4.046, Y 39.525, Z 16.150} C_DIS
   LIN {X 4.410, Y 38.336, Z 16.150} C_DIS
   LIN {X 4.481, Y 38.105, Z 16.150} C_DIS
   LIN {X 4.545, Y 37.884, Z 16.150} C_DIS
   LIN {X 5.014, Y 36.262, Z 16.150} C_DIS
   LIN {X 5.528, Y 34.343, Z 16.150} C_DIS
   LIN {X 5.734, Y 33.563, Z 16.150} C_DIS
   LIN {X 6.260, Y 31.348, Z 16.150} C_DIS
   LIN {X 6.484, Y 30.407, Z 16.150} C_DIS
   LIN {X 6.599, Y 29.868, Z 16.150} C_DIS
   LIN {X 6.872, Y 28.589, Z 16.150} C_DIS
   LIN {X 7.080, Y 27.503, Z 16.150} C_DIS
   LIN {X 7.425, Y 25.688, Z 16.150} C_DIS
   LIN {X 7.800, Y 23.287, Z 16.150} C_DIS
   LIN {X 8.142, Y 21.079, Z 16.150} C_DIS
   LIN {X 8.482, Y 18.218, Z 16.150} C_DIS
   LIN {X 8.620, Y 16.989, Z 16.150} C_DIS
   LIN {X 8.793, Y 14.756, Z 16.150} C_DIS
   LIN {X 8.967, Y 12.430, Z 16.150} C_DIS
   LIN {X 9.016, Y 11.092, Z 16.150} C_DIS
   LIN {X 9.115, Y 8.551, Z 16.150} C_DIS
   LIN {X 9.122, Y 5.826, Z 16.150} C_DIS
   LIN {X 9.036, Y 2.441, Z 16.150} C_DIS
   LIN {X 8.993, Y 0.883, Z 16.150} C_DIS
   LIN {X 8.893, Y -0.929, Z 16.150} C_DIS
   LIN {X 8.800, Y -2.112, Z 16.150}
   LaserEnd_Ext()
   LIN {X -11.280, Y -26.821, Z 16.150}
   LaserStart_Ext()
   LIN {X -11.280, Y -19.512, Z 16.150}
   LaserEnd_Ext()
   LIN {X -10.280, Y -17.568, Z 16.150}
   LaserStart_Ext()
   LIN {X -10.280, Y -28.294, Z 16.150}
   LaserEnd_Ext()
   LIN {X -9.280, Y -29.287, Z 16.150}
   LaserStart_Ext()
   LIN {X -9.280, Y -26.255, Z 16.150}
   LaserEnd_Ext()
   LIN {X -9.280, Y -20.066, Z 16.150}
   LaserStart_Ext()
   LIN {X -9.280, Y -15.797, Z 16.150}
   LaserEnd_Ext()
   LIN {X -8.280, Y -13.888, Z 16.150}
   LaserStart_Ext()
   LIN {X -8.280, Y -18.720, Z 16.150}
   LaserEnd_Ext()
   LIN {X -8.280, Y -27.520, Z 16.150}
   LaserStart_Ext()
   LIN {X -8.280, Y -29.988, Z 16.150}
   LaserEnd_Ext()
   LIN {X -7.280, Y -30.429, Z 16.150}
   LaserStart_Ext()
   LIN {X -7.280, Y -28.244, Z 16.150}
   LaserEnd_Ext()
   LIN {X -7.280, Y -18.021, Z 16.150}
   LaserStart_Ext()
   LIN {X -7.280, Y -11.773, Z 16.150}
   LaserEnd_Ext()
   LIN {X -6.280, Y -9.562, Z 16.150}
   LaserStart_Ext()
   LIN {X -6.280, Y -17.566, Z 16.150}
   LaserEnd_Ext()
   LIN {X -6.280, Y -28.719, Z 16.150}
   LaserStart_Ext()
   LIN {X -6.280, Y -30.759, Z 16.150}
   LaserEnd_Ext()
   LIN {X -5.280, Y -30.935, Z 16.150}
   LaserStart_Ext()
   LIN {X -5.280, Y -28.973, Z 16.150}
   LaserEnd_Ext()
   LIN {X -5.280, Y -17.166, Z 16.150}
   LaserStart_Ext()
   LIN {X -5.280, Y -7.006, Z 16.150}
   LaserEnd_Ext()
   LIN {X -4.280, Y -4.272, Z 16.150}
   LaserStart_Ext()
   LIN {X -4.280, Y -17.196, Z 16.150}
   LaserEnd_Ext()
   LIN {X -4.280, Y -29.053, Z 16.150}
   LaserStart_Ext()
   LIN {X -4.280, Y -31.007, Z 16.150}
   LaserEnd_Ext()
   LIN {X -3.280, Y -30.883, Z 16.150}
   LaserStart_Ext()
   LIN {X -3.280, Y -28.942, Z 16.150}
   LaserEnd_Ext()
   LIN {X -3.280, Y -17.330, Z 16.150}
   LaserStart_Ext()
   LIN {X -3.280, Y -0.902, Z 16.150}
   LaserEnd_Ext()
   LIN {X -2.280, Y 39.893, Z 16.150}
   LaserStart_Ext()
   LIN {X -2.280, Y 36.050, Z 16.150}
   LaserEnd_Ext()
   LIN {X -2.280, Y 2.733, Z 16.150}
   LaserStart_Ext()
   LIN {X -2.280, Y -17.468, Z 16.150}
